LIN {X 0,Y 164.587,Z 329.946,A -85,B 0,C 180,E1 -23658.193,E2 -23658.193} C_VEL
LIN {X 0,Y 167.282,Z 320.465,A -85,B 0,C 180,E1 -23660.938,E2 -23660.938} C_VEL
LIN {X 0,Y 169.157,Z 312.465,A -85,B 0,C 180,E1 -23662.842,E2 -23662.842} C_VEL
LIN {X 0,Y 167.967,Z 302.982,A -85,B 0,C 180,E1 -23665.202,E2 -23665.202} C_VEL
LIN {X 0,Y 166.059,Z 292.21,A -85,B 0,C 180,E1 -23667.577,E2 -23667.577} C_VEL
LIN {X 0,Y 163.931,Z 284.61,A -85,B 0,C 180,E1 -23669.159,E2 -23669.159} C_VEL
LIN {X 0,Y 159.909,Z 273.473,A -85,B 0,C 180,E1 -23671.379,E2 -23671.379} C_VEL
LIN {X 0,Y 158.08,Z 269.283,A -85,B 0,C 180,E1 -23672.192,E2 -23672.192} C_VEL
LIN {X 0,Y 157.989,Z 268.806,A -85,B 0,C 180,E1 -23672.393,E2 -23672.393} C_VEL
LIN {X 0,Y 157.793,Z 268.827,A -85,B 0,C 180,E1 -23677.681,E2 -23677.681} C_VEL
LIN {X 0,Y 157.67,Z 268.846,A -85,B 0,C 180,E1 -23681.32,E2 -23681.32} C_VEL
LIN {X 0,Y 157.48,Z 268.865,A -85,B 0,C 180,E1 -23685.534,E2 -23685.534} C_VEL
LIN {X 0,Y 157.408,Z 268.871,A -85,B 0,C 180,E1 -23690.93,E2 -23690.93} C_VEL
LIN {X 0,Y 157.312,Z 268.897,A -85,B 0,C 180,E1 -23696.692,E2 -23696.692} C_VEL
LIN {X 0,Y 157.277,Z 268.897,A -85,B 0,C 180,E1 -23702.43,E2 -23702.43} C_VEL
LIN {X 0,Y 157.317,Z 268.892,A -85,B 0,C 180,E1 -23706.481,E2 -23706.481} C_VEL
LIN {X 0,Y 157.283,Z 268.893,A -85,B 0,C 180,E1 -23712.09,E2 -23712.09} C_VEL
LIN {X 0,Y 157.299,Z 268.885,A -85,B 0,C 180,E1 -23715.636,E2 -23715.636} C_VEL
LIN {X 0,Y 157.285,Z 268.887,A -85,B 0,C 180,E1 -23721.282,E2 -23721.282} C_VEL
LIN {X 0,Y 157.29,Z 268.867,A -85,B 0,C 180,E1 -23724.494,E2 -23724.494} C_VEL
LIN {X 0,Y 157.294,Z 268.877,A -85,B 0,C 180,E1 -23728.1,E2 -23728.1} C_VEL
LIN {X 0,Y 157.324,Z 268.886,A -85,B 0,C 180,E1 -23733.471,E2 -23733.471} C_VEL
LIN {X 0,Y 157.397,Z 268.851,A -85,B 0,C 180,E1 -23739.673,E2 -23739.673} C_VEL
LIN {X 0,Y 157.478,Z 268.864,A -85,B 0,C 180,E1 -23744.473,E2 -23744.473} C_VEL
LIN {X 0,Y 157.695,Z 268.837,A -85,B 0,C 180,E1 -23749.735,E2 -23749.735} C_VEL
LIN {X 0,Y 157.772,Z 268.814,A -85,B 0,C 180,E1 -23752.324,E2 -23752.324} C_VEL
LIN {X 0,Y 158.263,Z 268.771,A -85,B 0,C 180,E1 -23760.004,E2 -23760.004} C_VEL
LIN {X 0,Y 157.773,Z 268.811,A -85,B 0,C 180,E1 -23767.684,E2 -23767.684} C_VEL
LIN {X 0,Y 157.646,Z 268.843,A -85,B 0,C 180,E1 -23771.24,E2 -23771.24} C_VEL
LIN {X 0,Y 157.463,Z 268.868,A -85,B 0,C 180,E1 -23775.537,E2 -23775.537} C_VEL
LIN {X 0,Y 157.381,Z 268.875,A -85,B 0,C 180,E1 -23780.935,E2 -23780.935} C_VEL
LIN {X 0,Y 157.325,Z 268.88,A -85,B 0,C 180,E1 -23786.686,E2 -23786.686} C_VEL
LIN {X 0,Y 157.3,Z 268.891,A -85,B 0,C 180,E1 -23792.426,E2 -23792.426} C_VEL
LIN {X 0,Y 157.397,Z 268.894,A -85,B 0,C 180,E1 -23794.706,E2 -23794.706} C_VEL
LIN {X 0,Y 158.075,Z 272.801,A -85,B 0,C 180,E1 -23800.899,E2 -23800.899} C_VEL
LIN {X 0,Y 158.59,Z 275.681,A -85,B 0,C 180,E1 -23805.162,E2 -23805.162} C_VEL
LIN {X 0,Y 159.285,Z 279.509,A -85,B 0,C 180,E1 -23810.551,E2 -23810.551} C_VEL
LIN {X 0,Y 161.987,Z 290.335,A -85,B 0,C 180,E1 -23812.106,E2 -23812.106} C_VEL
LIN {X 0,Y 163.705,Z 303.35,A -85,B 0,C 180,E1 -23814.073,E2 -23814.073} C_VEL
LIN {X 0,Y 164.706,Z 315.537,A -85,B 0,C 180,E1 -23816.306,E2 -23816.306} C_VEL
LIN {X 0,Y 165.012,Z 327.489,A -85,B 0,C 180,E1 -23818.905,E2 -23818.905} C_VEL
LIN {X 0,Y 164.792,Z 338.132,A -85,B 0,C 180,E1 -23821.673,E2 -23821.673} C_VEL
LIN {X 0,Y 164.335,Z 342.575,A -85,B 0,C 180,E1 -23822.972,E2 -23822.972} C_VEL
LIN {X 0,Y 161.587,Z 352.064,A -85,B 0,C 180,E1 -23826.068,E2 -23826.068} C_VEL
LIN {X 0,Y 159.321,Z 360.012,A -85,B 0,C 180,E1 -23829.333,E2 -23829.333} C_VEL
LIN {X 0,Y 157.38,Z 367.337,A -85,B 0,C 180,E1 -23833.123,E2 -23833.123} C_VEL
LIN {X 0,Y 155.955,Z 373.175,A -85,B 0,C 180,E1 -23836.976,E2 -23836.976} C_VEL
LIN {X 0,Y 155.267,Z 377.758,A -85,B 0,C 180,E1 -23840.882,E2 -23840.882} C_VEL
LIN {X 0,Y 155.188,Z 381.439,A -85,B 0,C 180,E1 -23845.115,E2 -23845.115} C_VEL
LIN {X 0,Y 155.179,Z 382.901,A -85,B 0,C 180,E1 -23847.402,E2 -23847.402} C_VEL
LIN {X 0,Y 155.293,Z 384.154,A -85,B 0,C 180,E1 -23849.997,E2 -23849.997} C_VEL
LIN {X 0,Y 154.993,Z 385.225,A -85,B 0,C 180,E1 -23853.948,E2 -23853.948} C_VEL
LIN {X 0,Y 155.003,Z 385.398,A -85,B 0,C 180,E1 -23857.815,E2 -23857.815} C_VEL
LIN {X 0,Y 155.909,Z 384.263,A -85,B 0,C 180,E1 -23863.023,E2 -23863.023} C_VEL
LIN {X 0,Y 158.117,Z 381.644,A -85,B 0,C 180,E1 -23868.125,E2 -23868.125} C_VEL
LIN {X 0,Y 161.641,Z 377.372,A -85,B 0,C 180,E1 -23873.033,E2 -23873.033} C_VEL
LIN {X 0,Y 164.907,Z 373.147,A -85,B 0,C 180,E1 -23876.488,E2 -23876.488} C_VEL
LIN {X 0,Y 169.712,Z 366.592,A -85,B 0,C 180,E1 -23880.481,E2 -23880.481} C_VEL
LIN {X 0,Y 174.548,Z 359.672,A -85,B 0,C 180,E1 -23883.614,E2 -23883.614} C_VEL
LIN {X 0,Y 177.754,Z 354.234,A -85,B 0,C 180,E1 -23885.672,E2 -23885.672} C_VEL
LIN {X 0,Y 180.555,Z 346.618,A -85,B 0,C 180,E1 -23888.517,E2 -23888.517} C_VEL
LIN {X 0,Y 182.546,Z 338.652,A -85,B 0,C 180,E1 -23891.297,E2 -23891.297} C_VEL
LIN {X 0,Y 183.154,Z 335.05,A -85,B 0,C 180,E1 -23892.533,E2 -23892.533} C_VEL
LIN {X 0,Y 183.282,Z 332.559,A -85,B 0,C 180,E1 -23893.482,E2 -23893.482} C_VEL
LIN {X 0,Y 182.549,Z 329.462,A -85,B 0,C 180,E1 -23895.048,E2 -23895.048} C_VEL
LIN {X 0,Y 180.077,Z 325.41,A -85,B 0,C 180,E1 -23897.863,E2 -23897.863} C_VEL
LIN {X 0,Y 177.491,Z 320.441,A -85,B 0,C 180,E1 -23901.38,E2 -23901.38} C_VEL
LIN {X 0,Y 176.191,Z 315.483,A -85,B 0,C 180,E1 -23904.536,E2 -23904.536} C_VEL
LIN {X 0,Y 175.099,Z 311.4,A -85,B 0,C 180,E1 -23907.441,E2 -23907.441} C_VEL
LIN {X 0,Y 173.845,Z 307.667,A -85,B 0,C 180,E1 -23910.976,E2 -23910.976} C_VEL
LIN {X 0,Y 173.102,Z 305.534,A -85,B 0,C 180,E1 -23913.47,E2 -23913.47} C_VEL
LIN {X 0,Y 172.072,Z 302.924,A -85,B 0,C 180,E1 -23918.429,E2 -23918.429} C_VEL
LIN {X 0,Y 171.945,Z 302.092,A -85,B 0,C 180,E1 -23920.91,E2 -23920.91} C_VEL
LIN {X 0,Y 171.99,Z 301.706,A -85,B 0,C 180,E1 -23923.375,E2 -23923.375} C_VEL
LIN {X 0,Y 172.781,Z 301.961,A -85,B 0,C 180,E1 -23928.262,E2 -23928.262} C_VEL
LIN {X 0,Y 173.598,Z 302.45,A -85,B 0,C 180,E1 -23930.677,E2 -23930.677} C_VEL
LIN {X 0,Y 174.34,Z 303.735,A -85,B 0,C 180,E1 -23933.05,E2 -23933.05} C_VEL
LIN {X 0,Y 176.32,Z 307.197,A -85,B 0,C 180,E1 -23937.712,E2 -23937.712} C_VEL
LIN {X 0,Y 177.681,Z 311.262,A -85,B 0,C 180,E1 -23941.13,E2 -23941.13} C_VEL
LIN {X 0,Y 179.166,Z 315.803,A -85,B 0,C 180,E1 -23944.496,E2 -23944.496} C_VEL
LIN {X 0,Y 180.317,Z 322.298,A -85,B 0,C 180,E1 -23948.401,E2 -23948.401} C_VEL
LIN {X 0,Y 180.587,Z 327.752,A -85,B 0,C 180,E1 -23951.217,E2 -23951.217} C_VEL
LIN {X 0,Y 179.946,Z 333.811,A -85,B 0,C 180,E1 -23954.125,E2 -23954.125} C_VEL
LIN {X 0,Y 179.697,Z 335.138,A -85,B 0,C 180,E1 -23954.723,E2 -23954.723} C_VEL
LIN {X 0,Y 176.11,Z 341.104,A -85,B 0,C 180,E1 -23956.721,E2 -23956.721} C_VEL
LIN {X 0,Y 171.383,Z 347.887,A -85,B 0,C 180,E1 -23959.416,E2 -23959.416} C_VEL
LIN {X 0,Y 165.978,Z 354.738,A -85,B 0,C 180,E1 -23962.962,E2 -23962.962} C_VEL
LIN {X 0,Y 160.917,Z 360.293,A -85,B 0,C 180,E1 -23966.898,E2 -23966.898} C_VEL
LIN {X 0,Y 156.483,Z 364.662,A -85,B 0,C 180,E1 -23971.429,E2 -23971.429} C_VEL
LIN {X 0,Y 153.937,Z 366.84,A -85,B 0,C 180,E1 -23974.741,E2 -23974.741} C_VEL
LIN {X 0,Y 151.811,Z 368.316,A -85,B 0,C 180,E1 -23978.098,E2 -23978.098} C_VEL
LIN {X 0,Y 150.161,Z 369.099,A -85,B 0,C 180,E1 -23981.513,E2 -23981.513} C_VEL
LIN {X 0,Y 148.898,Z 369.276,A -85,B 0,C 180,E1 -23985.066,E2 -23985.066} C_VEL
LIN {X 0,Y 147.965,Z 368.552,A -85,B 0,C 180,E1 -23989.453,E2 -23989.453} C_VEL
LIN {X 0,Y 147.657,Z 366.732,A -85,B 0,C 180,E1 -23994.004,E2 -23994.004} C_VEL
LIN {X 0,Y 148.074,Z 363.667,A -85,B 0,C 180,E1 -23998.677,E2 -23998.677} C_VEL
LIN {X 0,Y 149.184,Z 359.094,A -85,B 0,C 180,E1 -24003.508,E2 -24003.508} C_VEL
LIN {X 0,Y 150.768,Z 353.195,A -85,B 0,C 180,E1 -24008.107,E2 -24008.107} C_VEL
LIN {X 0,Y 153.045,Z 345.665,A -85,B 0,C 180,E1 -24012.526,E2 -24012.526} C_VEL
LIN {X 0,Y 155.63,Z 337.437,A -85,B 0,C 180,E1 -24016.288,E2 -24016.288} C_VEL
LIN {X 0,Y 158.101,Z 329.265,A -85,B 0,C 180,E1 -24019.267,E2 -24019.267} C_VEL
LIN {X 0,Y 161.001,Z 319.261,A -85,B 0,C 180,E1 -24022.162,E2 -24022.162} C_VEL
LIN {X 0,Y 162.417,Z 313.83,A -85,B 0,C 180,E1 -24023.48,E2 -24023.48} C_VEL
LIN {X 0,Y 161.154,Z 303.303,A -85,B 0,C 180,E1 -24026.252,E2 -24026.252} C_VEL
LIN {X 0,Y 159.17,Z 292.055,A -85,B 0,C 180,E1 -24028.864,E2 -24028.864} C_VEL
LIN {X 0,Y 155.263,Z 279.895,A -85,B 0,C 180,E1 -24031.541,E2 -24031.541} C_VEL
LIN {X 0,Y 152.291,Z 273.166,A -85,B 0,C 180,E1 -24033.025,E2 -24033.025} C_VEL
LIN {X 0,Y 150.941,Z 270.501,A -85,B 0,C 180,E1 -24033.632,E2 -24033.632} C_VEL
LIN {X 0,Y 150.772,Z 269.701,A -85,B 0,C 180,E1 -24033.845,E2 -24033.845} C_VEL
LIN {X 0,Y 150.728,Z 269.706,A -85,B 0,C 180,E1 -24038.044,E2 -24038.044} C_VEL
LIN {X 0,Y 150.601,Z 269.727,A -85,B 0,C 180,E1 -24041.505,E2 -24041.505} C_VEL
LIN {X 0,Y 150.389,Z 269.753,A -85,B 0,C 180,E1 -24046.286,E2 -24046.286} C_VEL
LIN {X 0,Y 150.381,Z 269.747,A -85,B 0,C 180,E1 -24050.836,E2 -24050.836} C_VEL
LIN {X 0,Y 150.241,Z 269.774,A -85,B 0,C 180,E1 -24057.289,E2 -24057.289} C_VEL
LIN {X 0,Y 150.217,Z 269.775,A -85,B 0,C 180,E1 -24062.642,E2 -24062.642} C_VEL
LIN {X 0,Y 150.228,Z 269.773,A -85,B 0,C 180,E1 -24067.461,E2 -24067.461} C_VEL
LIN {X 0,Y 150.224,Z 269.772,A -85,B 0,C 180,E1 -24071.544,E2 -24071.544} C_VEL
LIN {X 0,Y 150.249,Z 269.763,A -85,B 0,C 180,E1 -24075.448,E2 -24075.448} C_VEL
LIN {X 0,Y 150.227,Z 269.771,A -85,B 0,C 180,E1 -24079.09,E2 -24079.09} C_VEL
LIN {X 0,Y 150.234,Z 269.758,A -85,B 0,C 180,E1 -24082.685,E2 -24082.685} C_VEL
LIN {X 0,Y 150.218,Z 269.754,A -85,B 0,C 180,E1 -24087.371,E2 -24087.371} C_VEL
LIN {X 0,Y 150.246,Z 269.769,A -85,B 0,C 180,E1 -24092.723,E2 -24092.723} C_VEL
LIN {X 0,Y 150.354,Z 269.728,A -85,B 0,C 180,E1 -24099.213,E2 -24099.213} C_VEL
LIN {X 0,Y 150.383,Z 269.743,A -85,B 0,C 180,E1 -24103.72,E2 -24103.72} C_VEL
LIN {X 0,Y 150.618,Z 269.72,A -85,B 0,C 180,E1 -24109.247,E2 -24109.247} C_VEL
LIN {X 0,Y 150.709,Z 269.694,A -85,B 0,C 180,E1 -24111.962,E2 -24111.962} C_VEL
LIN {X 0,Y 151.223,Z 269.648,A -85,B 0,C 180,E1 -24120.004,E2 -24120.004} C_VEL
LIN {X 0,Y 150.695,Z 269.692,A -85,B 0,C 180,E1 -24128.047,E2 -24128.047} C_VEL
LIN {X 0,Y 150.587,Z 269.723,A -85,B 0,C 180,E1 -24131.44,E2 -24131.44} C_VEL
LIN {X 0,Y 150.371,Z 269.749,A -85,B 0,C 180,E1 -24136.29,E2 -24136.29} C_VEL
LIN {X 0,Y 150.362,Z 269.749,A -85,B 0,C 180,E1 -24140.795,E2 -24140.795} C_VEL
LIN {X 0,Y 150.255,Z 269.758,A -85,B 0,C 180,E1 -24147.284,E2 -24147.284} C_VEL
LIN {X 0,Y 150.255,Z 269.769,A -85,B 0,C 180,E1 -24152.651,E2 -24152.651} C_VEL
LIN {X 0,Y 150.365,Z 269.919,A -85,B 0,C 180,E1 -24154.526,E2 -24154.526} C_VEL
LIN {X 0,Y 151.01,Z 273.603,A -85,B 0,C 180,E1 -24160.664,E2 -24160.664} C_VEL
LIN {X 0,Y 151.645,Z 277.021,A -85,B 0,C 180,E1 -24165.955,E2 -24165.955} C_VEL
LIN {X 0,Y 152.064,Z 279.225,A -85,B 0,C 180,E1 -24169.04,E2 -24169.04} C_VEL
LIN {X 0,Y 152.993,Z 282.356,A -85,B 0,C 180,E1 -24169.507,E2 -24169.507} C_VEL
LIN {X 0,Y 155.105,Z 289.087,A -85,B 0,C 180,E1 -24170.624,E2 -24170.624} C_VEL
LIN {X 0,Y 156.73,Z 300.075,A -85,B 0,C 180,E1 -24172.371,E2 -24172.371} C_VEL
LIN {X 0,Y 157.918,Z 313.502,A -85,B 0,C 180,E1 -24174.863,E2 -24174.863} C_VEL
LIN {X 0,Y 158.22,Z 324.032,A -85,B 0,C 180,E1 -24177.176,E2 -24177.176} C_VEL
LIN {X 0,Y 158.076,Z 334.837,A -85,B 0,C 180,E1 -24179.986,E2 -24179.986} C_VEL
LIN {X 0,Y 157.685,Z 341.88,A -85,B 0,C 180,E1 -24182.094,E2 -24182.094} C_VEL
LIN {X 0,Y 154.776,Z 351.62,A -85,B 0,C 180,E1 -24185.386,E2 -24185.386} C_VEL
LIN {X 0,Y 152.252,Z 360.086,A -85,B 0,C 180,E1 -24189.036,E2 -24189.036} C_VEL
LIN {X 0,Y 150.256,Z 367.318,A -85,B 0,C 180,E1 -24192.999,E2 -24192.999} C_VEL
LIN {X 0,Y 149.006,Z 372.176,A -85,B 0,C 180,E1 -24196.357,E2 -24196.357} C_VEL
LIN {X 0,Y 148.239,Z 376.889,A -85,B 0,C 180,E1 -24200.446,E2 -24200.446} C_VEL
LIN {X 0,Y 148.124,Z 380.923,A -85,B 0,C 180,E1 -24205.166,E2 -24205.166} C_VEL
LIN {X 0,Y 148.228,Z 383.57,A -85,B 0,C 180,E1 -24209.997,E2 -24209.997} C_VEL
LIN {X 0,Y 147.924,Z 384.692,A -85,B 0,C 180,E1 -24213.809,E2 -24213.809} C_VEL
LIN {X 0,Y 147.953,Z 384.999,A -85,B 0,C 180,E1 -24218.19,E2 -24218.19} C_VEL
LIN {X 0,Y 148.971,Z 383.993,A -85,B 0,C 180,E1 -24223.641,E2 -24223.641} C_VEL
LIN {X 0,Y 151.355,Z 381.5,A -85,B 0,C 180,E1 -24228.965,E2 -24228.965} C_VEL
LIN {X 0,Y 154.044,Z 378.581,A -85,B 0,C 180,E1 -24232.815,E2 -24232.815} C_VEL
LIN {X 0,Y 157.454,Z 374.705,A -85,B 0,C 180,E1 -24236.507,E2 -24236.507} C_VEL
LIN {X 0,Y 161.364,Z 369.808,A -85,B 0,C 180,E1 -24240.054,E2 -24240.054} C_VEL
LIN {X 0,Y 166.955,Z 362.635,A -85,B 0,C 180,E1 -24243.898,E2 -24243.898} C_VEL
LIN {X 0,Y 171.297,Z 356.332,A -85,B 0,C 180,E1 -24246.503,E2 -24246.503} C_VEL
LIN {X 0,Y 174.417,Z 349.2,A -85,B 0,C 180,E1 -24249.351,E2 -24249.351} C_VEL
LIN {X 0,Y 176.905,Z 340.935,A -85,B 0,C 180,E1 -24252.48,E2 -24252.48} C_VEL
LIN {X 0,Y 178.724,Z 331.575,A -85,B 0,C 180,E1 -24255.885,E2 -24255.885} C_VEL
LIN {X 0,Y 178.953,Z 328.046,A -85,B 0,C 180,E1 -24257.271,E2 -24257.271} C_VEL
LIN {X 0,Y 177.746,Z 321.515,A -85,B 0,C 180,E1 -24260.751,E2 -24260.751} C_VEL
LIN {X 0,Y 177.491,Z 320.441,A -85,B 0,C 180,E1 -24261.38,E2 -24261.38} C_VEL
LIN {X 0,Y 176.414,Z 318.23,A -85,B 0,C 180,E1 -24263.116,E2 -24263.116} C_VEL
LIN {X 0,Y 174.799,Z 316.982,A -85,B 0,C 180,E1 -24264.942,E2 -24264.942} C_VEL
LIN {X 0,Y 171.436,Z 315.517,A -85,B 0,C 180,E1 -24268.756,E2 -24268.756} C_VEL
LIN {X 0,Y 170.376,Z 314.318,A -85,B 0,C 180,E1 -24270.707,E2 -24270.707} C_VEL
LIN {X 0,Y 170.201,Z 313.727,A -85,B 0,C 180,E1 -24271.352,E2 -24271.352} C_VEL
LIN {X 0,Y 169.873,Z 312.361,A -85,B 0,C 180,E1 -24272.925,E2 -24272.925} C_VEL
LIN {X 0,Y 169.205,Z 310.428,A -85,B 0,C 180,E1 -24276.027,E2 -24276.027} C_VEL
LIN {X 0,Y 168.8,Z 308.583,A -85,B 0,C 180,E1 -24280.54,E2 -24280.54} C_VEL
LIN {X 0,Y 168.834,Z 308.087,A -85,B 0,C 180,E1 -24283.21,E2 -24283.21} C_VEL
LIN {X 0,Y 169.516,Z 308.242,A -85,B 0,C 180,E1 -24288.032,E2 -24288.032} C_VEL
LIN {X 0,Y 170.259,Z 308.715,A -85,B 0,C 180,E1 -24290.493,E2 -24290.493} C_VEL
LIN {X 0,Y 170.835,Z 309.926,A -85,B 0,C 180,E1 -24292.907,E2 -24292.907} C_VEL
LIN {X 0,Y 172.491,Z 313.333,A -85,B 0,C 180,E1 -24297.661,E2 -24297.661} C_VEL
LIN {X 0,Y 173.9,Z 318.689,A -85,B 0,C 180,E1 -24302.313,E2 -24302.313} C_VEL
LIN {X 0,Y 174.586,Z 321.794,A -85,B 0,C 180,E1 -24304.614,E2 -24304.614} C_VEL
LIN {X 0,Y 175.157,Z 327.207,A -85,B 0,C 180,E1 -24308.069,E2 -24308.069} C_VEL
LIN {X 0,Y 175.059,Z 331.387,A -85,B 0,C 180,E1 -24310.404,E2 -24310.404} C_VEL
LIN {X 0,Y 174.112,Z 337.154,A -85,B 0,C 180,E1 -24313.377,E2 -24313.377} C_VEL
LIN {X 0,Y 171.784,Z 340.942,A -85,B 0,C 180,E1 -24314.726,E2 -24314.726} C_VEL
LIN {X 0,Y 166.076,Z 348.63,A -85,B 0,C 180,E1 -24317.804,E2 -24317.804} C_VEL
LIN {X 0,Y 160.681,Z 355.089,A -85,B 0,C 180,E1 -24321.218,E2 -24321.218} C_VEL
LIN {X 0,Y 155.332,Z 360.626,A -85,B 0,C 180,E1 -24325.196,E2 -24325.196} C_VEL
LIN {X 0,Y 150.443,Z 365.062,A -85,B 0,C 180,E1 -24329.903,E2 -24329.903} C_VEL
LIN {X 0,Y 146.304,Z 368.15,A -85,B 0,C 180,E1 -24335.257,E2 -24335.257} C_VEL
LIN {X 0,Y 143.923,Z 369.385,A -85,B 0,C 180,E1 -24339.4,E2 -24339.4} C_VEL
LIN {X 0,Y 142.14,Z 369.717,A -85,B 0,C 180,E1 -24343.799,E2 -24343.799} C_VEL
LIN {X 0,Y 140.856,Z 368.721,A -85,B 0,C 180,E1 -24349.565,E2 -24349.565} C_VEL
LIN {X 0,Y 140.595,Z 366.413,A -85,B 0,C 180,E1 -24354.914,E2 -24354.914} C_VEL
LIN {X 0,Y 141.224,Z 362.743,A -85,B 0,C 180,E1 -24360.159,E2 -24360.159} C_VEL
LIN {X 0,Y 142.536,Z 357.639,A -85,B 0,C 180,E1 -24365.225,E2 -24365.225} C_VEL
LIN {X 0,Y 144.468,Z 351.073,A -85,B 0,C 180,E1 -24370.094,E2 -24370.094} C_VEL
LIN {X 0,Y 146.814,Z 343.775,A -85,B 0,C 180,E1 -24374.217,E2 -24374.217} C_VEL
LIN {X 0,Y 149.32,Z 335.946,A -85,B 0,C 180,E1 -24377.722,E2 -24377.722} C_VEL
LIN {X 0,Y 152.291,Z 326.599,A -85,B 0,C 180,E1 -24381.042,E2 -24381.042} C_VEL
LIN {X 0,Y 155.444,Z 315.832,A -85,B 0,C 180,E1 -24384.037,E2 -24384.037} C_VEL
LIN {X 0,Y 155.54,Z 312.991,A -85,B 0,C 180,E1 -24384.818,E2 -24384.818} C_VEL
LIN {X 0,Y 154.223,Z 302.636,A -85,B 0,C 180,E1 -24387.657,E2 -24387.657} C_VEL
LIN {X 0,Y 152.425,Z 293.007,A -85,B 0,C 180,E1 -24390.003,E2 -24390.003} C_VEL
LIN {X 0,Y 148.529,Z 280.926,A -85,B 0,C 180,E1 -24392.868,E2 -24392.868} C_VEL
LIN {X 0,Y 144.783,Z 273.65,A -85,B 0,C 180,E1 -24394.745,E2 -24394.745} C_VEL
LIN {X 0,Y 143.71,Z 271.131,A -85,B 0,C 180,E1 -24395.326,E2 -24395.326} C_VEL
LIN {X 0,Y 143.635,Z 270.59,A -85,B 0,C 180,E1 -24395.425,E2 -24395.425} C_VEL
LIN {X 0,Y 143.649,Z 270.586,A -85,B 0,C 180,E1 -24398.443,E2 -24398.443} C_VEL
LIN {X 0,Y 143.538,Z 270.606,A -85,B 0,C 180,E1 -24401.716,E2 -24401.716} C_VEL
LIN {X 0,Y 143.327,Z 270.636,A -85,B 0,C 180,E1 -24407.113,E2 -24407.113} C_VEL
LIN {X 0,Y 143.303,Z 270.626,A -85,B 0,C 180,E1 -24411.294,E2 -24411.294} C_VEL
LIN {X 0,Y 143.187,Z 270.652,A -85,B 0,C 180,E1 -24417.945,E2 -24417.945} C_VEL
LIN {X 0,Y 143.166,Z 270.649,A -85,B 0,C 180,E1 -24423.443,E2 -24423.443} C_VEL
LIN {X 0,Y 143.119,Z 270.653,A -85,B 0,C 180,E1 -24429.674,E2 -24429.674} C_VEL
LIN {X 0,Y 143.158,Z 270.652,A -85,B 0,C 180,E1 -24433.42,E2 -24433.42} C_VEL
LIN {X 0,Y 143.154,Z 270.652,A -85,B 0,C 180,E1 -24437.43,E2 -24437.43} C_VEL
LIN {X 0,Y 143.137,Z 270.647,A -85,B 0,C 180,E1 -24441.78,E2 -24441.78} C_VEL
LIN {X 0,Y 143.185,Z 270.628,A -85,B 0,C 180,E1 -24447.328,E2 -24447.328} C_VEL
LIN {X 0,Y 143.192,Z 270.648,A -85,B 0,C 180,E1 -24452.068,E2 -24452.068} C_VEL
LIN {X 0,Y 143.28,Z 270.61,A -85,B 0,C 180,E1 -24458.751,E2 -24458.751} C_VEL
LIN {X 0,Y 143.318,Z 270.619,A -85,B 0,C 180,E1 -24462.894,E2 -24462.894} C_VEL
LIN {X 0,Y 143.543,Z 270.601,A -85,B 0,C 180,E1 -24468.711,E2 -24468.711} C_VEL
LIN {X 0,Y 143.631,Z 270.578,A -85,B 0,C 180,E1 -24471.563,E2 -24471.563} C_VEL
LIN {X 0,Y 144.182,Z 270.525,A -85,B 0,C 180,E1 -24480.004,E2 -24480.004} C_VEL
LIN {X 0,Y 143.62,Z 270.574,A -85,B 0,C 180,E1 -24488.446,E2 -24488.446} C_VEL
LIN {X 0,Y 143.515,Z 270.605,A -85,B 0,C 180,E1 -24491.633,E2 -24491.633} C_VEL
LIN {X 0,Y 143.311,Z 270.622,A -85,B 0,C 180,E1 -24497.116,E2 -24497.116} C_VEL
LIN {X 0,Y 143.288,Z 270.631,A -85,B 0,C 180,E1 -24501.257,E2 -24501.257} C_VEL
LIN {X 0,Y 143.201,Z 270.636,A -85,B 0,C 180,E1 -24507.939,E2 -24507.939} C_VEL
LIN {X 0,Y 143.292,Z 270.771,A -85,B 0,C 180,E1 -24514.083,E2 -24514.083} C_VEL
LIN {X 0,Y 143.794,Z 273.837,A -85,B 0,C 180,E1 -24519.453,E2 -24519.453} C_VEL
LIN {X 0,Y 144.447,Z 277.118,A -85,B 0,C 180,E1 -24524.873,E2 -24524.873} C_VEL
LIN {X 0,Y 144.754,Z 278.666,A -85,B 0,C 180,E1 -24527.306,E2 -24527.306} C_VEL
LIN {X 0,Y 145.76,Z 281.86,A -85,B 0,C 180,E1 -24527.84,E2 -24527.84} C_VEL
LIN {X 0,Y 148.591,Z 289.961,A -85,B 0,C 180,E1 -24529.373,E2 -24529.373} C_VEL
LIN {X 0,Y 149.988,Z 298.506,A -85,B 0,C 180,E1 -24530.829,E2 -24530.829} C_VEL
LIN {X 0,Y 151.094,Z 311.014,A -85,B 0,C 180,E1 -24533.208,E2 -24533.208} C_VEL
LIN {X 0,Y 151.485,Z 322.367,A -85,B 0,C 180,E1 -24535.766,E2 -24535.766} C_VEL
LIN {X 0,Y 151.385,Z 332.946,A -85,B 0,C 180,E1 -24538.579,E2 -24538.579} C_VEL
LIN {X 0,Y 150.799,Z 342.181,A -85,B 0,C 180,E1 -24541.462,E2 -24541.462} C_VEL
LIN {X 0,Y 147.933,Z 351.262,A -85,B 0,C 180,E1 -24544.683,E2 -24544.683} C_VEL
LIN {X 0,Y 145.204,Z 360.149,A -85,B 0,C 180,E1 -24548.712,E2 -24548.712} C_VEL
LIN {X 0,Y 143.114,Z 367.28,A -85,B 0,C 180,E1 -24552.861,E2 -24552.861} C_VEL
LIN {X 0,Y 141.705,Z 372.94,A -85,B 0,C 180,E1 -24557.101,E2 -24557.101} C_VEL
LIN {X 0,Y 141.064,Z 377.381,A -85,B 0,C 180,E1 -24561.401,E2 -24561.401} C_VEL
LIN {X 0,Y 141.041,Z 380.459,A -85,B 0,C 180,E1 -24565.313,E2 -24565.313} C_VEL
LIN {X 0,Y 141.163,Z 382.984,A -85,B 0,C 180,E1 -24569.997,E2 -24569.997} C_VEL
LIN {X 0,Y 140.854,Z 384.076,A -85,B 0,C 180,E1 -24573.647,E2 -24573.647} C_VEL
LIN {X 0,Y 140.903,Z 384.563,A -85,B 0,C 180,E1 -24578.603,E2 -24578.603} C_VEL
LIN {X 0,Y 142.038,Z 383.729,A -85,B 0,C 180,E1 -24584.321,E2 -24584.321} C_VEL
LIN {X 0,Y 144.632,Z 381.352,A -85,B 0,C 180,E1 -24589.883,E2 -24589.883} C_VEL
LIN {X 0,Y 148.673,Z 377.454,A -85,B 0,C 180,E1 -24595.176,E2 -24595.176} C_VEL
LIN {X 0,Y 152.393,Z 373.399,A -85,B 0,C 180,E1 -24598.958,E2 -24598.958} C_VEL
LIN {X 0,Y 156.85,Z 368.288,A -85,B 0,C 180,E1 -24602.523,E2 -24602.523} C_VEL
LIN {X 0,Y 162.035,Z 361.974,A -85,B 0,C 180,E1 -24605.838,E2 -24605.838} C_VEL
LIN {X 0,Y 165.614,Z 356.974,A -85,B 0,C 180,E1 -24607.972,E2 -24607.972} C_VEL
LIN {X 0,Y 168.671,Z 350.734,A -85,B 0,C 180,E1 -24610.658,E2 -24610.658} C_VEL
LIN {X 0,Y 171.604,Z 342.195,A -85,B 0,C 180,E1 -24614.122,E2 -24614.122} C_VEL
LIN {X 0,Y 173.345,Z 335.147,A -85,B 0,C 180,E1 -24616.865,E2 -24616.865} C_VEL
LIN {X 0,Y 173.759,Z 332.024,A -85,B 0,C 180,E1 -24618.192,E2 -24618.192} C_VEL
LIN {X 0,Y 172.814,Z 325.374,A -85,B 0,C 180,E1 -24622.065,E2 -24622.065} C_VEL
LIN {X 0,Y 171.692,Z 319.866,A -85,B 0,C 180,E1 -24625.876,E2 -24625.876} C_VEL
LIN {X 0,Y 171.255,Z 317.352,A -85,B 0,C 180,E1 -24627.754,E2 -24627.754} C_VEL
LIN {X 0,Y 170.201,Z 313.727,A -85,B 0,C 180,E1 -24631.352,E2 -24631.352} C_VEL
LIN {X 0,Y 169.801,Z 312.828,A -85,B 0,C 180,E1 -24632.629,E2 -24632.629} C_VEL
LIN {X 0,Y 168.744,Z 312.582,A -85,B 0,C 180,E1 -24634.596,E2 -24634.596} C_VEL
LIN {X 0,Y 165.419,Z 314.586,A -85,B 0,C 180,E1 -24640.68,E2 -24640.68} C_VEL
LIN {X 0,Y 165.272,Z 314.522,A -85,B 0,C 180,E1 -24642.08,E2 -24642.08} C_VEL
LIN {X 0,Y 165.918,Z 314.358,A -85,B 0,C 180,E1 -24647.769,E2 -24647.769} C_VEL
LIN {X 0,Y 166.568,Z 314.77,A -85,B 0,C 180,E1 -24650.28,E2 -24650.28} C_VEL
LIN {X 0,Y 167.031,Z 315.932,A -85,B 0,C 180,E1 -24652.745,E2 -24652.745} C_VEL
LIN {X 0,Y 168.351,Z 319.262,A -85,B 0,C 180,E1 -24657.604,E2 -24657.604} C_VEL
LIN {X 0,Y 169.341,Z 324.47,A -85,B 0,C 180,E1 -24662.375,E2 -24662.375} C_VEL
LIN {X 0,Y 169.772,Z 329.295,A -85,B 0,C 180,E1 -24665.938,E2 -24665.938} C_VEL
LIN {X 0,Y 169.642,Z 333.895,A -85,B 0,C 180,E1 -24668.934,E2 -24668.934} C_VEL
LIN {X 0,Y 168.814,Z 338.214,A -85,B 0,C 180,E1 -24671.401,E2 -24671.401} C_VEL
LIN {X 0,Y 168.502,Z 339.377,A -85,B 0,C 180,E1 -24672.033,E2 -24672.033} C_VEL
LIN {X 0,Y 167.589,Z 340.967,A -85,B 0,C 180,E1 -24672.678,E2 -24672.678} C_VEL
LIN {X 0,Y 161.914,Z 348.265,A -85,B 0,C 180,E1 -24675.538,E2 -24675.538} C_VEL
LIN {X 0,Y 156.084,Z 354.892,A -85,B 0,C 180,E1 -24679,E2 -24679} C_VEL
LIN {X 0,Y 151.628,Z 359.331,A -85,B 0,C 180,E1 -24682.035,E2 -24682.035} C_VEL
LIN {X 0,Y 145.739,Z 364.527,A -85,B 0,C 180,E1 -24687.002,E2 -24687.002} C_VEL
LIN {X 0,Y 141.14,Z 367.849,A -85,B 0,C 180,E1 -24692.172,E2 -24692.172} C_VEL
LIN {X 0,Y 137.514,Z 369.746,A -85,B 0,C 180,E1 -24697.821,E2 -24697.821} C_VEL
LIN {X 0,Y 135.178,Z 370.111,A -85,B 0,C 180,E1 -24703.296,E2 -24703.296} C_VEL
LIN {X 0,Y 134.163,Z 369.573,A -85,B 0,C 180,E1 -24707.163,E2 -24707.163} C_VEL
LIN {X 0,Y 133.497,Z 367.956,A -85,B 0,C 180,E1 -24712.147,E2 -24712.147} C_VEL
LIN {X 0,Y 133.685,Z 365.173,A -85,B 0,C 180,E1 -24717.251,E2 -24717.251} C_VEL
LIN {X 0,Y 134.646,Z 360.933,A -85,B 0,C 180,E1 -24722.529,E2 -24722.529} C_VEL
LIN {X 0,Y 135.933,Z 356.247,A -85,B 0,C 180,E1 -24726.89,E2 -24726.89} C_VEL
LIN {X 0,Y 137.908,Z 349.952,A -85,B 0,C 180,E1 -24731.43,E2 -24731.43} C_VEL
LIN {X 0,Y 140.34,Z 342.753,A -85,B 0,C 180,E1 -24735.502,E2 -24735.502} C_VEL
LIN {X 0,Y 143.09,Z 334.555,A -85,B 0,C 180,E1 -24739.183,E2 -24739.183} C_VEL
LIN {X 0,Y 146.108,Z 325.285,A -85,B 0,C 180,E1 -24742.471,E2 -24742.471} C_VEL
LIN {X 0,Y 148.74,Z 316.659,A -85,B 0,C 180,E1 -24744.92,E2 -24744.92} C_VEL
LIN {X 0,Y 148.726,Z 313.206,A -85,B 0,C 180,E1 -24745.938,E2 -24745.938} C_VEL
LIN {X 0,Y 147.516,Z 303.077,A -85,B 0,C 180,E1 -24748.839,E2 -24748.839} C_VEL
LIN {X 0,Y 146.423,Z 296.64,A -85,B 0,C 180,E1 -24750.519,E2 -24750.519} C_VEL
LIN {X 0,Y 142.872,Z 284.784,A -85,B 0,C 180,E1 -24753.599,E2 -24753.599} C_VEL
LIN {X 0,Y 137.946,Z 274.891,A -85,B 0,C 180,E1 -24756.351,E2 -24756.351} C_VEL
LIN {X 0,Y 136.667,Z 272.174,A -85,B 0,C 180,E1 -24757.065,E2 -24757.065} C_VEL
LIN {X 0,Y 136.554,Z 271.475,A -85,B 0,C 180,E1 -24757.21,E2 -24757.21} C_VEL
LIN {X 0,Y 136.481,Z 271.485,A -85,B 0,C 180,E1 -24761.958,E2 -24761.958} C_VEL
LIN {X 0,Y 136.266,Z 271.517,A -85,B 0,C 180,E1 -24768.029,E2 -24768.029} C_VEL
LIN {X 0,Y 136.219,Z 271.507,A -85,B 0,C 180,E1 -24771.785,E2 -24771.785} C_VEL
LIN {X 0,Y 136.113,Z 271.532,A -85,B 0,C 180,E1 -24778.636,E2 -24778.636} C_VEL
LIN {X 0,Y 136.078,Z 271.534,A -85,B 0,C 180,E1 -24784.622,E2 -24784.622} C_VEL
LIN {X 0,Y 136.085,Z 271.529,A -85,B 0,C 180,E1 -24789.234,E2 -24789.234} C_VEL
LIN {X 0,Y 136.094,Z 271.531,A -85,B 0,C 180,E1 -24793.707,E2 -24793.707} C_VEL
LIN {X 0,Y 136.104,Z 271.53,A -85,B 0,C 180,E1 -24797.841,E2 -24797.841} C_VEL
LIN {X 0,Y 136.089,Z 271.525,A -85,B 0,C 180,E1 -24801.711,E2 -24801.711} C_VEL
LIN {X 0,Y 136.091,Z 271.502,A -85,B 0,C 180,E1 -24805.722,E2 -24805.722} C_VEL
LIN {X 0,Y 136.148,Z 271.526,A -85,B 0,C 180,E1 -24812.322,E2 -24812.322} C_VEL
LIN {X 0,Y 136.247,Z 271.484,A -85,B 0,C 180,E1 -24818.839,E2 -24818.839} C_VEL
LIN {X 0,Y 136.283,Z 271.505,A -85,B 0,C 180,E1 -24825.063,E2 -24825.063} C_VEL
LIN {X 0,Y 136.463,Z 271.485,A -85,B 0,C 180,E1 -24828.117,E2 -24828.117} C_VEL
LIN {X 0,Y 136.557,Z 271.462,A -85,B 0,C 180,E1 -24831.123,E2 -24831.123} C_VEL
LIN {X 0,Y 137.139,Z 271.402,A -85,B 0,C 180,E1 -24840.005,E2 -24840.005} C_VEL
LIN {X 0,Y 136.549,Z 271.456,A -85,B 0,C 180,E1 -24848.887,E2 -24848.887} C_VEL
LIN {X 0,Y 136.45,Z 271.486,A -85,B 0,C 180,E1 -24851.894,E2 -24851.894} C_VEL
LIN {X 0,Y 136.252,Z 271.496,A -85,B 0,C 180,E1 -24858.033,E2 -24858.033} C_VEL
LIN {X 0,Y 136.209,Z 271.515,A -85,B 0,C 180,E1 -24861.752,E2 -24861.752} C_VEL
LIN {X 0,Y 136.112,Z 271.521,A -85,B 0,C 180,E1 -24868.618,E2 -24868.618} C_VEL
LIN {X 0,Y 136.222,Z 271.624,A -85,B 0,C 180,E1 -24873.605,E2 -24873.605} C_VEL
LIN {X 0,Y 136.793,Z 274.88,A -85,B 0,C 180,E1 -24879.583,E2 -24879.583} C_VEL
LIN {X 0,Y 137.433,Z 278.178,A -85,B 0,C 180,E1 -24885.269,E2 -24885.269} C_VEL
LIN {X 0,Y 137.638,Z 279.235,A -85,B 0,C 180,E1 -24885.524,E2 -24885.524} C_VEL
LIN {X 0,Y 139.023,Z 282.414,A -85,B 0,C 180,E1 -24886.213,E2 -24886.213} C_VEL
LIN {X 0,Y 142.38,Z 291.903,A -85,B 0,C 180,E1 -24888.21,E2 -24888.21} C_VEL
LIN {X 0,Y 143.617,Z 299.832,A -85,B 0,C 180,E1 -24889.71,E2 -24889.71} C_VEL
LIN {X 0,Y 144.514,Z 311.961,A -85,B 0,C 180,E1 -24892.185,E2 -24892.185} C_VEL
LIN {X 0,Y 144.807,Z 323.611,A -85,B 0,C 180,E1 -24895,E2 -24895} C_VEL
LIN {X 0,Y 144.511,Z 334.334,A -85,B 0,C 180,E1 -24898.067,E2 -24898.067} C_VEL
LIN {X 0,Y 143.921,Z 342.441,A -85,B 0,C 180,E1 -24900.766,E2 -24900.766} C_VEL
LIN {X 0,Y 140.684,Z 352.149,A -85,B 0,C 180,E1 -24904.446,E2 -24904.446} C_VEL
LIN {X 0,Y 138.149,Z 360.19,A -85,B 0,C 180,E1 -24908.354,E2 -24908.354} C_VEL
LIN {X 0,Y 135.989,Z 367.201,A -85,B 0,C 180,E1 -24912.71,E2 -24912.71} C_VEL
LIN {X 0,Y 134.442,Z 373.593,A -85,B 0,C 180,E1 -24917.927,E2 -24917.927} C_VEL
LIN {X 0,Y 133.938,Z 377.777,A -85,B 0,C 180,E1 -24922.459,E2 -24922.459} C_VEL
LIN {X 0,Y 133.963,Z 380.853,A -85,B 0,C 180,E1 -24926.99,E2 -24926.99} C_VEL
LIN {X 0,Y 134.098,Z 382.339,A -85,B 0,C 180,E1 -24929.997,E2 -24929.997} C_VEL
LIN {X 0,Y 133.795,Z 383.461,A -85,B 0,C 180,E1 -24933.533,E2 -24933.533} C_VEL
LIN {X 0,Y 133.856,Z 384.127,A -85,B 0,C 180,E1 -24939.059,E2 -24939.059} C_VEL
LIN {X 0,Y 135.137,Z 383.434,A -85,B 0,C 180,E1 -24945.069,E2 -24945.069} C_VEL
LIN {X 0,Y 136.304,Z 382.527,A -85,B 0,C 180,E1 -24948.018,E2 -24948.018} C_VEL
LIN {X 0,Y 139.901,Z 379.544,A -85,B 0,C 180,E1 -24953.693,E2 -24953.693} C_VEL
LIN {X 0,Y 143.535,Z 376.269,A -85,B 0,C 180,E1 -24957.717,E2 -24957.717} C_VEL
LIN {X 0,Y 147.689,Z 372.018,A -85,B 0,C 180,E1 -24961.561,E2 -24961.561} C_VEL
LIN {X 0,Y 153.538,Z 365.696,A -85,B 0,C 180,E1 -24965.702,E2 -24965.702} C_VEL
LIN {X 0,Y 159.226,Z 358.945,A -85,B 0,C 180,E1 -24968.971,E2 -24968.971} C_VEL
LIN {X 0,Y 162.688,Z 352.868,A -85,B 0,C 180,E1 -24971.749,E2 -24971.749} C_VEL
LIN {X 0,Y 165.89,Z 344.992,A -85,B 0,C 180,E1 -24975.2,E2 -24975.2} C_VEL
LIN {X 0,Y 167.972,Z 338.45,A -85,B 0,C 180,E1 -24977.971,E2 -24977.971} C_VEL
LIN {X 0,Y 168.459,Z 335.773,A -85,B 0,C 180,E1 -24979.198,E2 -24979.198} C_VEL
LIN {X 0,Y 168.019,Z 330.33,A -85,B 0,C 180,E1 -24982.627,E2 -24982.627} C_VEL
LIN {X 0,Y 167.196,Z 324.614,A -85,B 0,C 180,E1 -24986.872,E2 -24986.872} C_VEL
LIN {X 0,Y 167.051,Z 322.891,A -85,B 0,C 180,E1 -24988.267,E2 -24988.267} C_VEL
LIN {X 0,Y 166.16,Z 318.764,A -85,B 0,C 180,E1 -24992.646,E2 -24992.646} C_VEL
LIN {X 0,Y 165.428,Z 315.919,A -85,B 0,C 180,E1 -24997.517,E2 -24997.517} C_VEL
LIN {X 0,Y 165.272,Z 314.522,A -85,B 0,C 180,E1 -25002.08,E2 -25002.08} C_VEL
LIN {X 0,Y 165.144,Z 314.725,A -85,B 0,C 180,E1 -25004.124,E2 -25004.124} C_VEL
LIN {X 0,Y 164.596,Z 315.933,A -85,B 0,C 180,E1 -25006.136,E2 -25006.136} C_VEL
LIN {X 0,Y 162.99,Z 320.905,A -85,B 0,C 180,E1 -25011.478,E2 -25011.478} C_VEL
LIN {X 0,Y 162.982,Z 321.895,A -85,B 0,C 180,E1 -25012.856,E2 -25012.856} C_VEL
LIN {X 0,Y 163.92,Z 324.961,A -85,B 0,C 180,E1 -25017.539,E2 -25017.539} C_VEL
LIN {X 0,Y 164.456,Z 330.035,A -85,B 0,C 180,E1 -25022.445,E2 -25022.445} C_VEL
LIN {X 0,Y 164.432,Z 334.686,A -85,B 0,C 180,E1 -25026.13,E2 -25026.13} C_VEL
LIN {X 0,Y 163.907,Z 338.368,A -85,B 0,C 180,E1 -25028.628,E2 -25028.628} C_VEL
LIN {X 0,Y 163.02,Z 341.491,A -85,B 0,C 180,E1 -25030.554,E2 -25030.554} C_VEL
LIN {X 0,Y 161.394,Z 343.885,A -85,B 0,C 180,E1 -25031.562,E2 -25031.562} C_VEL
LIN {X 0,Y 154.616,Z 351.749,A -85,B 0,C 180,E1 -25035.014,E2 -25035.014} C_VEL
LIN {X 0,Y 148.417,Z 357.951,A -85,B 0,C 180,E1 -25038.736,E2 -25038.736} C_VEL
LIN {X 0,Y 142.214,Z 363.304,A -85,B 0,C 180,E1 -25043.283,E2 -25043.283} C_VEL
LIN {X 0,Y 137.873,Z 366.505,A -85,B 0,C 180,E1 -25047.302,E2 -25047.302} C_VEL
LIN {X 0,Y 133.463,Z 369.135,A -85,B 0,C 180,E1 -25052.596,E2 -25052.596} C_VEL
LIN {X 0,Y 131.019,Z 370.18,A -85,B 0,C 180,E1 -25056.432,E2 -25056.432} C_VEL
LIN {X 0,Y 128.875,Z 370.56,A -85,B 0,C 180,E1 -25060.867,E2 -25060.867} C_VEL
LIN {X 0,Y 127.311,Z 370.064,A -85,B 0,C 180,E1 -25065.853,E2 -25065.853} C_VEL
LIN {X 0,Y 126.42,Z 368.037,A -85,B 0,C 180,E1 -25072.305,E2 -25072.305} C_VEL
LIN {X 0,Y 126.711,Z 364.647,A -85,B 0,C 180,E1 -25078.292,E2 -25078.292} C_VEL
LIN {X 0,Y 127.869,Z 360.014,A -85,B 0,C 180,E1 -25083.919,E2 -25083.919} C_VEL
LIN {X 0,Y 129.404,Z 354.845,A -85,B 0,C 180,E1 -25088.605,E2 -25088.605} C_VEL
LIN {X 0,Y 131.831,Z 347.598,A -85,B 0,C 180,E1 -25093.638,E2 -25093.638} C_VEL
LIN {X 0,Y 134.704,Z 339.532,A -85,B 0,C 180,E1 -25097.957,E2 -25097.957} C_VEL
LIN {X 0,Y 138.024,Z 329.949,A -85,B 0,C 180,E1 -25101.954,E2 -25101.954} C_VEL
LIN {X 0,Y 141.081,Z 320.511,A -85,B 0,C 180,E1 -25105.015,E2 -25105.015} C_VEL
LIN {X 0,Y 142.218,Z 316.595,A -85,B 0,C 180,E1 -25106.112,E2 -25106.112} C_VEL
LIN {X 0,Y 141.19,Z 306.069,A -85,B 0,C 180,E1 -25109.389,E2 -25109.389} C_VEL
LIN {X 0,Y 139.896,Z 298.32,A -85,B 0,C 180,E1 -25111.625,E2 -25111.625} C_VEL
LIN {X 0,Y 136.968,Z 288.086,A -85,B 0,C 180,E1 -25114.49,E2 -25114.49} C_VEL
LIN {X 0,Y 130.927,Z 275.787,A -85,B 0,C 180,E1 -25118.242,E2 -25118.242} C_VEL
LIN {X 0,Y 129.62,Z 272.89,A -85,B 0,C 180,E1 -25119.069,E2 -25119.069} C_VEL
LIN {X 0,Y 129.505,Z 272.346,A -85,B 0,C 180,E1 -25119.274,E2 -25119.274} C_VEL
LIN {X 0,Y 129.385,Z 272.368,A -85,B 0,C 180,E1 -25122.552,E2 -25122.552} C_VEL
LIN {X 0,Y 129.178,Z 272.398,A -85,B 0,C 180,E1 -25129.056,E2 -25129.056} C_VEL
LIN {X 0,Y 129.128,Z 272.391,A -85,B 0,C 180,E1 -25132.398,E2 -25132.398} C_VEL
LIN {X 0,Y 129.029,Z 272.416,A -85,B 0,C 180,E1 -25139.379,E2 -25139.379} C_VEL
LIN {X 0,Y 129.02,Z 272.416,A -85,B 0,C 180,E1 -25145.215,E2 -25145.215} C_VEL
LIN {X 0,Y 129.01,Z 272.414,A -85,B 0,C 180,E1 -25150.826,E2 -25150.826} C_VEL
LIN {X 0,Y 129.022,Z 272.407,A -85,B 0,C 180,E1 -25155.087,E2 -25155.087} C_VEL
LIN {X 0,Y 129.012,Z 272.414,A -85,B 0,C 180,E1 -25159.704,E2 -25159.704} C_VEL
LIN {X 0,Y 129.023,Z 272.382,A -85,B 0,C 180,E1 -25164.797,E2 -25164.797} C_VEL
LIN {X 0,Y 129.034,Z 272.409,A -85,B 0,C 180,E1 -25170.653,E2 -25170.653} C_VEL
LIN {X 0,Y 129.111,Z 272.38,A -85,B 0,C 180,E1 -25177.608,E2 -25177.608} C_VEL
LIN {X 0,Y 129.162,Z 272.366,A -85,B 0,C 180,E1 -25180.95,E2 -25180.95} C_VEL
LIN {X 0,Y 129.404,Z 272.365,A -85,B 0,C 180,E1 -25187.861,E2 -25187.861} C_VEL
LIN {X 0,Y 129.485,Z 272.346,A -85,B 0,C 180,E1 -25190.634,E2 -25190.634} C_VEL
LIN {X 0,Y 130.094,Z 272.279,A -85,B 0,C 180,E1 -25200.005,E2 -25200.005} C_VEL
LIN {X 0,Y 129.475,Z 272.339,A -85,B 0,C 180,E1 -25209.377,E2 -25209.377} C_VEL
LIN {X 0,Y 129.354,Z 272.372,A -85,B 0,C 180,E1 -25212.557,E2 -25212.557} C_VEL
LIN {X 0,Y 129.163,Z 272.378,A -85,B 0,C 180,E1 -25219.06,E2 -25219.06} C_VEL
LIN {X 0,Y 129.119,Z 272.401,A -85,B 0,C 180,E1 -25222.401,E2 -25222.401} C_VEL
LIN {X 0,Y 129.047,Z 272.404,A -85,B 0,C 180,E1 -25229.376,E2 -25229.376} C_VEL
LIN {X 0,Y 129.171,Z 272.396,A -85,B 0,C 180,E1 -25232.968,E2 -25232.968} C_VEL
LIN {X 0,Y 129.639,Z 275.238,A -85,B 0,C 180,E1 -25238.573,E2 -25238.573} C_VEL
LIN {X 0,Y 130.143,Z 277.802,A -85,B 0,C 180,E1 -25243.252,E2 -25243.252} C_VEL
LIN {X 0,Y 131.156,Z 280.969,A -85,B 0,C 180,E1 -25243.894,E2 -25243.894} C_VEL
LIN {X 0,Y 132.328,Z 283.66,A -85,B 0,C 180,E1 -25244.549,E2 -25244.549} C_VEL
LIN {X 0,Y 135.542,Z 292.079,A -85,B 0,C 180,E1 -25246.551,E2 -25246.551} C_VEL
LIN {X 0,Y 136.911,Z 297.477,A -85,B 0,C 180,E1 -25247.745,E2 -25247.745} C_VEL
LIN {X 0,Y 137.896,Z 310.177,A -85,B 0,C 180,E1 -25250.451,E2 -25250.451} C_VEL
LIN {X 0,Y 138.164,Z 322.003,A -85,B 0,C 180,E1 -25253.402,E2 -25253.402} C_VEL
LIN {X 0,Y 137.783,Z 333.292,A -85,B 0,C 180,E1 -25256.744,E2 -25256.744} C_VEL
LIN {X 0,Y 137.042,Z 342.564,A -85,B 0,C 180,E1 -25259.996,E2 -25259.996} C_VEL
LIN {X 0,Y 133.764,Z 352.066,A -85,B 0,C 180,E1 -25263.797,E2 -25263.797} C_VEL
LIN {X 0,Y 131.1,Z 360.151,A -85,B 0,C 180,E1 -25267.957,E2 -25267.957} C_VEL
LIN {X 0,Y 128.884,Z 367.073,A -85,B 0,C 180,E1 -25272.544,E2 -25272.544} C_VEL
LIN {X 0,Y 127.483,Z 372.605,A -85,B 0,C 180,E1 -25277.257,E2 -25277.257} C_VEL
LIN {X 0,Y 126.888,Z 376.924,A -85,B 0,C 180,E1 -25282.038,E2 -25282.038} C_VEL
LIN {X 0,Y 126.886,Z 380.129,A -85,B 0,C 180,E1 -25286.822,E2 -25286.822} C_VEL
LIN {X 0,Y 127.033,Z 381.677,A -85,B 0,C 180,E1 -25289.997,E2 -25289.997} C_VEL
LIN {X 0,Y 126.749,Z 382.854,A -85,B 0,C 180,E1 -25293.497,E2 -25293.497} C_VEL
LIN {X 0,Y 126.834,Z 383.691,A -85,B 0,C 180,E1 -25299.566,E2 -25299.566} C_VEL
LIN {X 0,Y 128.246,Z 383.121,A -85,B 0,C 180,E1 -25305.899,E2 -25305.899} C_VEL
LIN {X 0,Y 131.325,Z 381.1,A -85,B 0,C 180,E1 -25311.997,E2 -25311.997} C_VEL
LIN {X 0,Y 135.927,Z 377.483,A -85,B 0,C 180,E1 -25317.729,E2 -25317.729} C_VEL
LIN {X 0,Y 140.112,Z 373.726,A -85,B 0,C 180,E1 -25321.778,E2 -25321.778} C_VEL
LIN {X 0,Y 145.085,Z 368.953,A -85,B 0,C 180,E1 -25325.538,E2 -25325.538} C_VEL
LIN {X 0,Y 151.826,Z 361.915,A -85,B 0,C 180,E1 -25329.527,E2 -25329.527} C_VEL
LIN {X 0,Y 154.615,Z 358.39,A -85,B 0,C 180,E1 -25331.227,E2 -25331.227} C_VEL
LIN {X 0,Y 158.129,Z 352.17,A -85,B 0,C 180,E1 -25334.267,E2 -25334.267} C_VEL
LIN {X 0,Y 161.441,Z 344.682,A -85,B 0,C 180,E1 -25337.733,E2 -25337.733} C_VEL
LIN {X 0,Y 162.93,Z 340.404,A -85,B 0,C 180,E1 -25339.678,E2 -25339.678} C_VEL
LIN {X 0,Y 163.09,Z 336.971,A -85,B 0,C 180,E1 -25341.881,E2 -25341.881} C_VEL
LIN {X 0,Y 162.775,Z 331.652,A -85,B 0,C 180,E1 -25345.851,E2 -25345.851} C_VEL
LIN {X 0,Y 162.564,Z 328.261,A -85,B 0,C 180,E1 -25348.745,E2 -25348.745} C_VEL
LIN {X 0,Y 162.056,Z 324.618,A -85,B 0,C 180,E1 -25352.794,E2 -25352.794} C_VEL
LIN {X 0,Y 161.548,Z 322.198,A -85,B 0,C 180,E1 -25356.946,E2 -25356.946} C_VEL
LIN {X 0,Y 161.475,Z 321.124,A -85,B 0,C 180,E1 -25359.62,E2 -25359.62} C_VEL
LIN {X 0,Y 161.523,Z 320.337,A -85,B 0,C 180,E1 -25363.174,E2 -25363.174} C_VEL
LIN {X 0,Y 161.987,Z 320.287,A -85,B 0,C 180,E1 -25367.467,E2 -25367.467} C_VEL
LIN {X 0,Y 162.567,Z 320.624,A -85,B 0,C 180,E1 -25370.038,E2 -25370.038} C_VEL
LIN {X 0,Y 162.982,Z 321.895,A -85,B 0,C 180,E1 -25372.856,E2 -25372.856} C_VEL
LIN {X 0,Y 162.886,Z 323.668,A -85,B 0,C 180,E1 -25374.839,E2 -25374.839} C_VEL
LIN {X 0,Y 162.243,Z 326.222,A -85,B 0,C 180,E1 -25376.716,E2 -25376.716} C_VEL
LIN {X 0,Y 159.511,Z 334.155,A -85,B 0,C 180,E1 -25381.642,E2 -25381.642} C_VEL
LIN {X 0,Y 159.184,Z 335.822,A -85,B 0,C 180,E1 -25382.958,E2 -25382.958} C_VEL
LIN {X 0,Y 158.699,Z 339.892,A -85,B 0,C 180,E1 -25386.352,E2 -25386.352} C_VEL
LIN {X 0,Y 157.744,Z 343.179,A -85,B 0,C 180,E1 -25388.658,E2 -25388.658} C_VEL
LIN {X 0,Y 156.821,Z 344.922,A -85,B 0,C 180,E1 -25389.636,E2 -25389.636} C_VEL
LIN {X 0,Y 149.62,Z 352.693,A -85,B 0,C 180,E1 -25393.131,E2 -25393.131} C_VEL
LIN {X 0,Y 142.631,Z 359.17,A -85,B 0,C 180,E1 -25397.191,E2 -25397.191} C_VEL
LIN {X 0,Y 136.207,Z 364.199,A -85,B 0,C 180,E1 -25401.766,E2 -25401.766} C_VEL
LIN {X 0,Y 132.201,Z 366.934,A -85,B 0,C 180,E1 -25405.352,E2 -25405.352} C_VEL
LIN {X 0,Y 128.381,Z 369.074,A -85,B 0,C 180,E1 -25409.511,E2 -25409.511} C_VEL
LIN {X 0,Y 125.007,Z 370.478,A -85,B 0,C 180,E1 -25414.202,E2 -25414.202} C_VEL
LIN {X 0,Y 122.373,Z 370.984,A -85,B 0,C 180,E1 -25419.171,E2 -25419.171} C_VEL
LIN {X 0,Y 120.264,Z 370.363,A -85,B 0,C 180,E1 -25425.477,E2 -25425.477} C_VEL
LIN {X 0,Y 119.513,Z 369.111,A -85,B 0,C 180,E1 -25429.851,E2 -25429.851} C_VEL
LIN {X 0,Y 119.338,Z 366.522,A -85,B 0,C 180,E1 -25435.525,E2 -25435.525} C_VEL
LIN {X 0,Y 120.282,Z 361.98,A -85,B 0,C 180,E1 -25442.136,E2 -25442.136} C_VEL
LIN {X 0,Y 121.784,Z 356.919,A -85,B 0,C 180,E1 -25447.404,E2 -25447.404} C_VEL
LIN {X 0,Y 124.033,Z 350.254,A -85,B 0,C 180,E1 -25452.697,E2 -25452.697} C_VEL
LIN {X 0,Y 126.71,Z 342.966,A -85,B 0,C 180,E1 -25457.185,E2 -25457.185} C_VEL
LIN {X 0,Y 129.986,Z 334.059,A -85,B 0,C 180,E1 -25461.452,E2 -25461.452} C_VEL
LIN {X 0,Y 133.675,Z 323.527,A -85,B 0,C 180,E1 -25465.318,E2 -25465.318} C_VEL
LIN {X 0,Y 135.479,Z 317.865,A -85,B 0,C 180,E1 -25467.029,E2 -25467.029} C_VEL
LIN {X 0,Y 134.685,Z 307.752,A -85,B 0,C 180,E1 -25470.377,E2 -25470.377} C_VEL
LIN {X 0,Y 133.64,Z 301.056,A -85,B 0,C 180,E1 -25472.433,E2 -25472.433} C_VEL
LIN {X 0,Y 130.832,Z 290.941,A -85,B 0,C 180,E1 -25475.547,E2 -25475.547} C_VEL
LIN {X 0,Y 125.621,Z 279.963,A -85,B 0,C 180,E1 -25479.259,E2 -25479.259} C_VEL
LIN {X 0,Y 123.779,Z 276.623,A -85,B 0,C 180,E1 -25480.415,E2 -25480.415} C_VEL
LIN {X 0,Y 122.498,Z 273.991,A -85,B 0,C 180,E1 -25481.266,E2 -25481.266} C_VEL
LIN {X 0,Y 122.357,Z 273.245,A -85,B 0,C 180,E1 -25481.523,E2 -25481.523} C_VEL
LIN {X 0,Y 122.123,Z 273.275,A -85,B 0,C 180,E1 -25486.726,E2 -25486.726} C_VEL
LIN {X 0,Y 122.06,Z 273.272,A -85,B 0,C 180,E1 -25492.906,E2 -25492.906} C_VEL
LIN {X 0,Y 121.955,Z 273.298,A -85,B 0,C 180,E1 -25497.457,E2 -25497.457} C_VEL
LIN {X 0,Y 121.907,Z 273.305,A -85,B 0,C 180,E1 -25501.259,E2 -25501.259} C_VEL
LIN {X 0,Y 121.933,Z 273.299,A -85,B 0,C 180,E1 -25506.213,E2 -25506.213} C_VEL
LIN {X 0,Y 121.939,Z 273.296,A -85,B 0,C 180,E1 -25511.482,E2 -25511.482} C_VEL
LIN {X 0,Y 121.94,Z 273.297,A -85,B 0,C 180,E1 -25518.531,E2 -25518.531} C_VEL
LIN {X 0,Y 121.975,Z 273.259,A -85,B 0,C 180,E1 -25524.824,E2 -25524.824} C_VEL
LIN {X 0,Y 121.943,Z 273.288,A -85,B 0,C 180,E1 -25529.833,E2 -25529.833} C_VEL
LIN {X 0,Y 121.986,Z 273.277,A -85,B 0,C 180,E1 -25536.222,E2 -25536.222} C_VEL
LIN {X 0,Y 122.051,Z 273.247,A -85,B 0,C 180,E1 -25539.794,E2 -25539.794} C_VEL
LIN {X 0,Y 122.249,Z 273.256,A -85,B 0,C 180,E1 -25546.711,E2 -25546.711} C_VEL
LIN {X 0,Y 122.421,Z 273.227,A -85,B 0,C 180,E1 -25550.088,E2 -25550.088} C_VEL
LIN {X 0,Y 122.602,Z 273.193,A -85,B 0,C 180,E1 -25556.719,E2 -25556.719} C_VEL
LIN {X 0,Y 123.047,Z 273.157,A -85,B 0,C 180,E1 -25560.005,E2 -25560.005} C_VEL
LIN {X 0,Y 122.425,Z 273.211,A -85,B 0,C 180,E1 -25566.598,E2 -25566.598} C_VEL
LIN {X 0,Y 122.321,Z 273.248,A -85,B 0,C 180,E1 -25572.368,E2 -25572.368} C_VEL
LIN {X 0,Y 122.118,Z 273.263,A -85,B 0,C 180,E1 -25576.729,E2 -25576.729} C_VEL
LIN {X 0,Y 122.035,Z 273.284,A -85,B 0,C 180,E1 -25582.854,E2 -25582.854} C_VEL
LIN {X 0,Y 122.015,Z 273.285,A -85,B 0,C 180,E1 -25590.226,E2 -25590.226} C_VEL
LIN {X 0,Y 122.127,Z 273.334,A -85,B 0,C 180,E1 -25592.655,E2 -25592.655} C_VEL
LIN {X 0,Y 122.664,Z 276.438,A -85,B 0,C 180,E1 -25599.074,E2 -25599.074} C_VEL
LIN {X 0,Y 122.858,Z 277.302,A -85,B 0,C 180,E1 -25600.806,E2 -25600.806} C_VEL
LIN {X 0,Y 123.892,Z 280.53,A -85,B 0,C 180,E1 -25601.539,E2 -25601.539} C_VEL
LIN {X 0,Y 125.133,Z 283.12,A -85,B 0,C 180,E1 -25602.283,E2 -25602.283} C_VEL
LIN {X 0,Y 129.121,Z 293.431,A -85,B 0,C 180,E1 -25605.045,E2 -25605.045} C_VEL
LIN {X 0,Y 130.697,Z 299.486,A -85,B 0,C 180,E1 -25606.553,E2 -25606.553} C_VEL
LIN {X 0,Y 131.473,Z 311.864,A -85,B 0,C 180,E1 -25609.395,E2 -25609.395} C_VEL
LIN {X 0,Y 131.549,Z 323.416,A -85,B 0,C 180,E1 -25612.52,E2 -25612.52} C_VEL
LIN {X 0,Y 130.974,Z 334.78,A -85,B 0,C 180,E1 -25616.167,E2 -25616.167} C_VEL
LIN {X 0,Y 130.193,Z 342.687,A -85,B 0,C 180,E1 -25619.144,E2 -25619.144} C_VEL
LIN {X 0,Y 126.872,Z 351.965,A -85,B 0,C 180,E1 -25623.068,E2 -25623.068} C_VEL
LIN {X 0,Y 124.046,Z 360.093,A -85,B 0,C 180,E1 -25627.512,E2 -25627.512} C_VEL
LIN {X 0,Y 121.778,Z 366.945,A -85,B 0,C 180,E1 -25632.36,E2 -25632.36} C_VEL
LIN {X 0,Y 120.214,Z 373.223,A -85,B 0,C 180,E1 -25638.189,E2 -25638.189} C_VEL
LIN {X 0,Y 119.78,Z 377.295,A -85,B 0,C 180,E1 -25643.258,E2 -25643.258} C_VEL
LIN {X 0,Y 119.821,Z 379.399,A -85,B 0,C 180,E1 -25646.634,E2 -25646.634} C_VEL
LIN {X 0,Y 119.968,Z 381.004,A -85,B 0,C 180,E1 -25649.997,E2 -25649.997} C_VEL
LIN {X 0,Y 119.691,Z 382.139,A -85,B 0,C 180,E1 -25653.363,E2 -25653.363} C_VEL
LIN {X 0,Y 119.806,Z 383.245,A -85,B 0,C 180,E1 -25660.132,E2 -25660.132} C_VEL
LIN {X 0,Y 121.388,Z 382.808,A -85,B 0,C 180,E1 -25666.824,E2 -25666.824} C_VEL
LIN {X 0,Y 124.755,Z 380.932,A -85,B 0,C 180,E1 -25673.221,E2 -25673.221} C_VEL
LIN {X 0,Y 126.986,Z 379.444,A -85,B 0,C 180,E1 -25676.276,E2 -25676.276} C_VEL
LIN {X 0,Y 132.189,Z 375.504,A -85,B 0,C 180,E1 -25681.709,E2 -25681.709} C_VEL
LIN {X 0,Y 137.539,Z 370.945,A -85,B 0,C 180,E1 -25685.985,E2 -25685.985} C_VEL
LIN {X 0,Y 144.35,Z 364.593,A -85,B 0,C 180,E1 -25690.17,E2 -25690.17} C_VEL
LIN {X 0,Y 148.447,Z 360.265,A -85,B 0,C 180,E1 -25692.423,E2 -25692.423} C_VEL
LIN {X 0,Y 151.877,Z 355.122,A -85,B 0,C 180,E1 -25695.137,E2 -25695.137} C_VEL
LIN {X 0,Y 155.239,Z 348.809,A -85,B 0,C 180,E1 -25698.326,E2 -25698.326} C_VEL
LIN {X 0,Y 157.034,Z 344.88,A -85,B 0,C 180,E1 -25700.246,E2 -25700.246} C_VEL
LIN {X 0,Y 157.615,Z 342.906,A -85,B 0,C 180,E1 -25701.368,E2 -25701.368} C_VEL
LIN {X 0,Y 157.8,Z 338.614,A -85,B 0,C 180,E1 -25704.617,E2 -25704.617} C_VEL
LIN {X 0,Y 157.833,Z 333.619,A -85,B 0,C 180,E1 -25709.026,E2 -25709.026} C_VEL
LIN {X 0,Y 157.614,Z 329.85,A -85,B 0,C 180,E1 -25713.515,E2 -25713.515} C_VEL
LIN {X 0,Y 157.373,Z 328.258,A -85,B 0,C 180,E1 -25716.298,E2 -25716.298} C_VEL
LIN {X 0,Y 157.292,Z 326.867,A -85,B 0,C 180,E1 -25719.761,E2 -25719.761} C_VEL
LIN {X 0,Y 157.449,Z 326.035,A -85,B 0,C 180,E1 -25724.462,E2 -25724.462} C_VEL
LIN {X 0,Y 158.259,Z 326.29,A -85,B 0,C 180,E1 -25729.764,E2 -25729.764} C_VEL
LIN {X 0,Y 158.582,Z 327.372,A -85,B 0,C 180,E1 -25732.5,E2 -25732.5} C_VEL
LIN {X 0,Y 159.199,Z 330.429,A -85,B 0,C 180,E1 -25737.466,E2 -25737.466} C_VEL
LIN {X 0,Y 159.256,Z 334.002,A -85,B 0,C 180,E1 -25741.26,E2 -25741.26} C_VEL
LIN {X 0,Y 159.184,Z 335.822,A -85,B 0,C 180,E1 -25742.958,E2 -25742.958} C_VEL
LIN {X 0,Y 158.651,Z 337.651,A -85,B 0,C 180,E1 -25744.206,E2 -25744.206} C_VEL
LIN {X 0,Y 156.738,Z 340.969,A -85,B 0,C 180,E1 -25745.853,E2 -25745.853} C_VEL
LIN {X 0,Y 153.935,Z 344.57,A -85,B 0,C 180,E1 -25747.297,E2 -25747.297} C_VEL
LIN {X 0,Y 149.322,Z 349.412,A -85,B 0,C 180,E1 -25749.159,E2 -25749.159} C_VEL
LIN {X 0,Y 144.655,Z 353.82,A -85,B 0,C 180,E1 -25751.211,E2 -25751.211} C_VEL
LIN {X 0,Y 138.117,Z 359.484,A -85,B 0,C 180,E1 -25754.816,E2 -25754.816} C_VEL
LIN {X 0,Y 132.387,Z 363.74,A -85,B 0,C 180,E1 -25758.568,E2 -25758.568} C_VEL
LIN {X 0,Y 127.214,Z 367.044,A -85,B 0,C 180,E1 -25762.745,E2 -25762.745} C_VEL
LIN {X 0,Y 122.722,Z 369.404,A -85,B 0,C 180,E1 -25767.261,E2 -25767.261} C_VEL
LIN {X 0,Y 118.046,Z 371.129,A -85,B 0,C 180,E1 -25773.546,E2 -25773.546} C_VEL
LIN {X 0,Y 115.729,Z 371.418,A -85,B 0,C 180,E1 -25777.87,E2 -25777.87} C_VEL
LIN {X 0,Y 113.866,Z 371.041,A -85,B 0,C 180,E1 -25782.752,E2 -25782.752} C_VEL
LIN {X 0,Y 112.558,Z 369.669,A -85,B 0,C 180,E1 -25788.518,E2 -25788.518} C_VEL
LIN {X 0,Y 112.26,Z 366.554,A -85,B 0,C 180,E1 -25795.71,E2 -25795.71} C_VEL
LIN {X 0,Y 113.237,Z 361.96,A -85,B 0,C 180,E1 -25802.531,E2 -25802.531} C_VEL
LIN {X 0,Y 114.979,Z 356.384,A -85,B 0,C 180,E1 -25808.489,E2 -25808.489} C_VEL
LIN {X 0,Y 117.208,Z 350.14,A -85,B 0,C 180,E1 -25813.593,E2 -25813.593} C_VEL
LIN {X 0,Y 119.963,Z 342.983,A -85,B 0,C 180,E1 -25818.171,E2 -25818.171} C_VEL
LIN {X 0,Y 123.399,Z 333.968,A -85,B 0,C 180,E1 -25822.641,E2 -25822.641} C_VEL
LIN {X 0,Y 126.773,Z 324.792,A -85,B 0,C 180,E1 -25826.178,E2 -25826.178} C_VEL
LIN {X 0,Y 128.831,Z 318.065,A -85,B 0,C 180,E1 -25828.36,E2 -25828.36} C_VEL
LIN {X 0,Y 128.026,Z 307.769,A -85,B 0,C 180,E1 -25831.968,E2 -25831.968} C_VEL
LIN {X 0,Y 126.817,Z 301.456,A -85,B 0,C 180,E1 -25834.109,E2 -25834.109} C_VEL
LIN {X 0,Y 125.013,Z 294.462,A -85,B 0,C 180,E1 -25836.459,E2 -25836.459} C_VEL
LIN {X 0,Y 119.801,Z 283.169,A -85,B 0,C 180,E1 -25840.63,E2 -25840.63} C_VEL
LIN {X 0,Y 116.779,Z 277.677,A -85,B 0,C 180,E1 -25842.779,E2 -25842.779} C_VEL
LIN {X 0,Y 115.364,Z 275.144,A -85,B 0,C 180,E1 -25843.777,E2 -25843.777} C_VEL
LIN {X 0,Y 115.143,Z 274.134,A -85,B 0,C 180,E1 -25844.135,E2 -25844.135} C_VEL
LIN {X 0,Y 115.005,Z 274.149,A -85,B 0,C 180,E1 -25851.514,E2 -25851.514} C_VEL
LIN {X 0,Y 114.874,Z 274.183,A -85,B 0,C 180,E1 -25855.361,E2 -25855.361} C_VEL
LIN {X 0,Y 114.864,Z 274.183,A -85,B 0,C 180,E1 -25861.075,E2 -25861.075} C_VEL
LIN {X 0,Y 114.844,Z 274.181,A -85,B 0,C 180,E1 -25867.736,E2 -25867.736} C_VEL
LIN {X 0,Y 114.862,Z 274.178,A -85,B 0,C 180,E1 -25872.766,E2 -25872.766} C_VEL
LIN {X 0,Y 114.867,Z 274.176,A -85,B 0,C 180,E1 -25877.708,E2 -25877.708} C_VEL
LIN {X 0,Y 114.854,Z 274.16,A -85,B 0,C 180,E1 -25882.706,E2 -25882.706} C_VEL
LIN {X 0,Y 114.869,Z 274.163,A -85,B 0,C 180,E1 -25888.939,E2 -25888.939} C_VEL
LIN {X 0,Y 114.949,Z 274.151,A -85,B 0,C 180,E1 -25896.514,E2 -25896.514} C_VEL
LIN {X 0,Y 115.02,Z 274.134,A -85,B 0,C 180,E1 -25902.217,E2 -25902.217} C_VEL
LIN {X 0,Y 115.258,Z 274.127,A -85,B 0,C 180,E1 -25907.337,E2 -25907.337} C_VEL
LIN {X 0,Y 115.371,Z 274.083,A -85,B 0,C 180,E1 -25913.008,E2 -25913.008} C_VEL
LIN {X 0,Y 115.999,Z 274.034,A -85,B 0,C 180,E1 -25920.005,E2 -25920.005} C_VEL
LIN {X 0,Y 115.367,Z 274.088,A -85,B 0,C 180,E1 -25927.004,E2 -25927.004} C_VEL
LIN {X 0,Y 115.258,Z 274.128,A -85,B 0,C 180,E1 -25932.662,E2 -25932.662} C_VEL
LIN {X 0,Y 115.021,Z 274.14,A -85,B 0,C 180,E1 -25937.794,E2 -25937.794} C_VEL
LIN {X 0,Y 114.958,Z 274.168,A -85,B 0,C 180,E1 -25943.496,E2 -25943.496} C_VEL
LIN {X 0,Y 115.045,Z 274.155,A -85,B 0,C 180,E1 -25952.078,E2 -25952.078} C_VEL
LIN {X 0,Y 115.532,Z 277.078,A -85,B 0,C 180,E1 -25958.093,E2 -25958.093} C_VEL
LIN {X 0,Y 116.808,Z 280.499,A -85,B 0,C 180,E1 -25959.031,E2 -25959.031} C_VEL
LIN {X 0,Y 117.883,Z 282.601,A -85,B 0,C 180,E1 -25959.725,E2 -25959.725} C_VEL
LIN {X 0,Y 120.916,Z 289.724,A -85,B 0,C 180,E1 -25961.875,E2 -25961.875} C_VEL
LIN {X 0,Y 123.77,Z 298.295,A -85,B 0,C 180,E1 -25964.376,E2 -25964.376} C_VEL
LIN {X 0,Y 124.706,Z 303.372,A -85,B 0,C 180,E1 -25965.722,E2 -25965.722} C_VEL
LIN {X 0,Y 125.055,Z 314.904,A -85,B 0,C 180,E1 -25968.67,E2 -25968.67} C_VEL
LIN {X 0,Y 124.863,Z 326.092,A -85,B 0,C 180,E1 -25972.006,E2 -25972.006} C_VEL
LIN {X 0,Y 124.009,Z 337.282,A -85,B 0,C 180,E1 -25975.965,E2 -25975.965} C_VEL
LIN {X 0,Y 123.404,Z 342.763,A -85,B 0,C 180,E1 -25978.207,E2 -25978.207} C_VEL
LIN {X 0,Y 120.128,Z 351.467,A -85,B 0,C 180,E1 -25982.09,E2 -25982.09} C_VEL
LIN {X 0,Y 117.032,Z 359.978,A -85,B 0,C 180,E1 -25987.021,E2 -25987.021} C_VEL
LIN {X 0,Y 114.685,Z 366.765,A -85,B 0,C 180,E1 -25992.154,E2 -25992.154} C_VEL
LIN {X 0,Y 113.255,Z 372.184,A -85,B 0,C 180,E1 -25997.452,E2 -25997.452} C_VEL
LIN {X 0,Y 112.728,Z 376.4,A -85,B 0,C 180,E1 -26002.834,E2 -26002.834} C_VEL
LIN {X 0,Y 112.766,Z 378.604,A -85,B 0,C 180,E1 -26006.423,E2 -26006.423} C_VEL
LIN {X 0,Y 112.905,Z 380.317,A -85,B 0,C 180,E1 -26009.996,E2 -26009.996} C_VEL
LIN {X 0,Y 112.611,Z 381.513,A -85,B 0,C 180,E1 -26013.575,E2 -26013.575} C_VEL
LIN {X 0,Y 112.807,Z 382.749,A -85,B 0,C 180,E1 -26020.768,E2 -26020.768} C_VEL
LIN {X 0,Y 114.568,Z 382.501,A -85,B 0,C 180,E1 -26027.858,E2 -26027.858} C_VEL
LIN {X 0,Y 118.235,Z 380.767,A -85,B 0,C 180,E1 -26034.584,E2 -26034.584} C_VEL
LIN {X 0,Y 123.483,Z 377.564,A -85,B 0,C 180,E1 -26040.809,E2 -26040.809} C_VEL
LIN {X 0,Y 130.011,Z 372.708,A -85,B 0,C 180,E1 -26046.482,E2 -26046.482} C_VEL
LIN {X 0,Y 135.815,Z 367.929,A -85,B 0,C 180,E1 -26050.3,E2 -26050.3} C_VEL
LIN {X 0,Y 142.271,Z 362.007,A -85,B 0,C 180,E1 -26053.751,E2 -26053.751} C_VEL
LIN {X 0,Y 145.811,Z 357.508,A -85,B 0,C 180,E1 -26056.298,E2 -26056.298} C_VEL
LIN {X 0,Y 149.7,Z 351.268,A -85,B 0,C 180,E1 -26059.716,E2 -26059.716} C_VEL
LIN {X 0,Y 151.801,Z 347.226,A -85,B 0,C 180,E1 -26061.907,E2 -26061.907} C_VEL
LIN {X 0,Y 152.35,Z 344.507,A -85,B 0,C 180,E1 -26063.969,E2 -26063.969} C_VEL
LIN {X 0,Y 152.707,Z 340.337,A -85,B 0,C 180,E1 -26067.752,E2 -26067.752} C_VEL
LIN {X 0,Y 152.866,Z 338.427,A -85,B 0,C 180,E1 -26069.616,E2 -26069.616} C_VEL
LIN {X 0,Y 152.885,Z 336.005,A -85,B 0,C 180,E1 -26072.629,E2 -26072.629} C_VEL
LIN {X 0,Y 152.796,Z 333.496,A -85,B 0,C 180,E1 -26076.908,E2 -26076.908} C_VEL
LIN {X 0,Y 152.828,Z 332.049,A -85,B 0,C 180,E1 -26081.218,E2 -26081.218} C_VEL
LIN {X 0,Y 153.228,Z 331.539,A -85,B 0,C 180,E1 -26086.738,E2 -26086.738} C_VEL
LIN {X 0,Y 153.674,Z 331.73,A -85,B 0,C 180,E1 -26089.455,E2 -26089.455} C_VEL
LIN {X 0,Y 153.917,Z 332.599,A -85,B 0,C 180,E1 -26092.123,E2 -26092.123} C_VEL
LIN {X 0,Y 154.017,Z 333.94,A -85,B 0,C 180,E1 -26094.76,E2 -26094.76} C_VEL
LIN {X 0,Y 154.2,Z 335.624,A -85,B 0,C 180,E1 -26097.384,E2 -26097.384} C_VEL
LIN {X 0,Y 153.909,Z 339.056,A -85,B 0,C 180,E1 -26101.304,E2 -26101.304} C_VEL
LIN {X 0,Y 153.124,Z 343.253,A -85,B 0,C 180,E1 -26105.263,E2 -26105.263} C_VEL
LIN {X 0,Y 152.209,Z 345.801,A -85,B 0,C 180,E1 -26107.291,E2 -26107.291} C_VEL
LIN {X 0,Y 151.51,Z 346.924,A -85,B 0,C 180,E1 -26107.995,E2 -26107.995} C_VEL
LIN {X 0,Y 144.655,Z 353.82,A -85,B 0,C 180,E1 -26111.211,E2 -26111.211} C_VEL
LIN {X 0,Y 141.053,Z 356.753,A -85,B 0,C 180,E1 -26112.688,E2 -26112.688} C_VEL
LIN {X 0,Y 133.84,Z 361.229,A -85,B 0,C 180,E1 -26114.841,E2 -26114.841} C_VEL
LIN {X 0,Y 126.662,Z 365.01,A -85,B 0,C 180,E1 -26117.338,E2 -26117.338} C_VEL
LIN {X 0,Y 123.22,Z 366.767,A -85,B 0,C 180,E1 -26119.359,E2 -26119.359} C_VEL
LIN {X 0,Y 117.293,Z 369.75,A -85,B 0,C 180,E1 -26124.792,E2 -26124.792} C_VEL
LIN {X 0,Y 113.109,Z 371.239,A -85,B 0,C 180,E1 -26129.8,E2 -26129.8} C_VEL
LIN {X 0,Y 109.748,Z 371.84,A -85,B 0,C 180,E1 -26135.186,E2 -26135.186} C_VEL
LIN {X 0,Y 107.285,Z 371.525,A -85,B 0,C 180,E1 -26140.917,E2 -26140.917} C_VEL
LIN {X 0,Y 105.488,Z 369.825,A -85,B 0,C 180,E1 -26148.228,E2 -26148.228} C_VEL
LIN {X 0,Y 105.172,Z 366.732,A -85,B 0,C 180,E1 -26155.558,E2 -26155.558} C_VEL
LIN {X 0,Y 106.046,Z 362.392,A -85,B 0,C 180,E1 -26162.365,E2 -26162.365} C_VEL
LIN {X 0,Y 107.948,Z 356.535,A -85,B 0,C 180,E1 -26169.022,E2 -26169.022} C_VEL
LIN {X 0,Y 110.317,Z 350.212,A -85,B 0,C 180,E1 -26174.457,E2 -26174.457} C_VEL
LIN {X 0,Y 113.226,Z 343,A -85,B 0,C 180,E1 -26179.272,E2 -26179.272} C_VEL
LIN {X 0,Y 116.866,Z 333.879,A -85,B 0,C 180,E1 -26183.962,E2 -26183.962} C_VEL
LIN {X 0,Y 120.784,Z 323.65,A -85,B 0,C 180,E1 -26187.989,E2 -26187.989} C_VEL
LIN {X 0,Y 122.063,Z 320.008,A -85,B 0,C 180,E1 -26189.179,E2 -26189.179} C_VEL
LIN {X 0,Y 121.905,Z 313.601,A -85,B 0,C 180,E1 -26191.646,E2 -26191.646} C_VEL
LIN {X 0,Y 121.364,Z 307.646,A -85,B 0,C 180,E1 -26193.809,E2 -26193.809} C_VEL
LIN {X 0,Y 119.272,Z 298.413,A -85,B 0,C 180,E1 -26197.196,E2 -26197.196} C_VEL
LIN {X 0,Y 114.73,Z 287.849,A -85,B 0,C 180,E1 -26201.477,E2 -26201.477} C_VEL
LIN {X 0,Y 110.786,Z 280.534,A -85,B 0,C 180,E1 -26204.703,E2 -26204.703} C_VEL
LIN {X 0,Y 108.298,Z 276.379,A -85,B 0,C 180,E1 -26206.614,E2 -26206.614} C_VEL
LIN {X 0,Y 107.981,Z 275.038,A -85,B 0,C 180,E1 -26207.033,E2 -26207.033} C_VEL
LIN {X 0,Y 107.866,Z 275.049,A -85,B 0,C 180,E1 -26214.209,E2 -26214.209} C_VEL
LIN {X 0,Y 107.794,Z 275.062,A -85,B 0,C 180,E1 -26222.063,E2 -26222.063} C_VEL
LIN {X 0,Y 107.751,Z 275.06,A -85,B 0,C 180,E1 -26228.502,E2 -26228.502} C_VEL
LIN {X 0,Y 107.766,Z 275.054,A -85,B 0,C 180,E1 -26235.843,E2 -26235.843} C_VEL
LIN {X 0,Y 107.754,Z 275.053,A -85,B 0,C 180,E1 -26241.512,E2 -26241.512} C_VEL
LIN {X 0,Y 107.811,Z 275.039,A -85,B 0,C 180,E1 -26248.574,E2 -26248.574} C_VEL
LIN {X 0,Y 107.913,Z 275.021,A -85,B 0,C 180,E1 -26257.005,E2 -26257.005} C_VEL
LIN {X 0,Y 108.038,Z 275.022,A -85,B 0,C 180,E1 -26264.924,E2 -26264.924} C_VEL
LIN {X 0,Y 108.263,Z 274.996,A -85,B 0,C 180,E1 -26268.776,E2 -26268.776} C_VEL
LIN {X 0,Y 108.45,Z 274.949,A -85,B 0,C 180,E1 -26276.29,E2 -26276.29} C_VEL
LIN {X 0,Y 108.948,Z 274.912,A -85,B 0,C 180,E1 -26280.006,E2 -26280.006} C_VEL
LIN {X 0,Y 108.307,Z 274.965,A -85,B 0,C 180,E1 -26287.463,E2 -26287.463} C_VEL
LIN {X 0,Y 108.179,Z 275.01,A -85,B 0,C 180,E1 -26292.953,E2 -26292.953} C_VEL
LIN {X 0,Y 107.914,Z 275.023,A -85,B 0,C 180,E1 -26299.01,E2 -26299.01} C_VEL
LIN {X 0,Y 107.869,Z 275.049,A -85,B 0,C 180,E1 -26304.188,E2 -26304.188} C_VEL
LIN {X 0,Y 108.003,Z 275.123,A -85,B 0,C 180,E1 -26311.87,E2 -26311.87} C_VEL
LIN {X 0,Y 108.176,Z 276.34,A -85,B 0,C 180,E1 -26314.777,E2 -26314.777} C_VEL
LIN {X 0,Y 109.186,Z 279.473,A -85,B 0,C 180,E1 -26315.698,E2 -26315.698} C_VEL
LIN {X 0,Y 110.773,Z 282.269,A -85,B 0,C 180,E1 -26316.836,E2 -26316.836} C_VEL
LIN {X 0,Y 114.255,Z 290.44,A -85,B 0,C 180,E1 -26319.663,E2 -26319.663} C_VEL
LIN {X 0,Y 117.69,Z 300.609,A -85,B 0,C 180,E1 -26322.968,E2 -26322.968} C_VEL
LIN {X 0,Y 118.538,Z 305.036,A -85,B 0,C 180,E1 -26324.285,E2 -26324.285} C_VEL
LIN {X 0,Y 118.656,Z 316.204,A -85,B 0,C 180,E1 -26327.375,E2 -26327.375} C_VEL
LIN {X 0,Y 118.299,Z 326.151,A -85,B 0,C 180,E1 -26330.57,E2 -26330.57} C_VEL
LIN {X 0,Y 117.296,Z 337.293,A -85,B 0,C 180,E1 -26334.777,E2 -26334.777} C_VEL
LIN {X 0,Y 116.624,Z 342.747,A -85,B 0,C 180,E1 -26337.152,E2 -26337.152} C_VEL
LIN {X 0,Y 113.226,Z 351.392,A -85,B 0,C 180,E1 -26341.242,E2 -26341.242} C_VEL
LIN {X 0,Y 110.01,Z 359.825,A -85,B 0,C 180,E1 -26346.463,E2 -26346.463} C_VEL
LIN {X 0,Y 107.583,Z 366.564,A -85,B 0,C 180,E1 -26351.919,E2 -26351.919} C_VEL
LIN {X 0,Y 105.983,Z 372.739,A -85,B 0,C 180,E1 -26358.521,E2 -26358.521} C_VEL
LIN {X 0,Y 105.658,Z 376.726,A -85,B 0,C 180,E1 -26364.272,E2 -26364.272} C_VEL
LIN {X 0,Y 105.843,Z 379.593,A -85,B 0,C 180,E1 -26369.996,E2 -26369.996} C_VEL
LIN {X 0,Y 105.534,Z 380.884,A -85,B 0,C 180,E1 -26373.815,E2 -26373.815} C_VEL
LIN {X 0,Y 105.808,Z 382.24,A -85,B 0,C 180,E1 -26381.49,E2 -26381.49} C_VEL
LIN {X 0,Y 107.796,Z 382.155,A -85,B 0,C 180,E1 -26389.021,E2 -26389.021} C_VEL
LIN {X 0,Y 111.78,Z 380.602,A -85,B 0,C 180,E1 -26396.107,E2 -26396.107} C_VEL
LIN {X 0,Y 117.406,Z 377.562,A -85,B 0,C 180,E1 -26402.594,E2 -26402.594} C_VEL
LIN {X 0,Y 122.489,Z 374.255,A -85,B 0,C 180,E1 -26407.042,E2 -26407.042} C_VEL
LIN {X 0,Y 128.38,Z 369.987,A -85,B 0,C 180,E1 -26411.061,E2 -26411.061} C_VEL
LIN {X 0,Y 136.149,Z 363.642,A -85,B 0,C 180,E1 -26415.212,E2 -26415.212} C_VEL
LIN {X 0,Y 139.135,Z 360.516,A -85,B 0,C 180,E1 -26417.086,E2 -26417.086} C_VEL
LIN {X 0,Y 143.28,Z 355.037,A -85,B 0,C 180,E1 -26420.378,E2 -26420.378} C_VEL
LIN {X 0,Y 145.851,Z 351.069,A -85,B 0,C 180,E1 -26422.657,E2 -26422.657} C_VEL
LIN {X 0,Y 146.726,Z 348.66,A -85,B 0,C 180,E1 -26424.511,E2 -26424.511} C_VEL
LIN {X 0,Y 147.483,Z 344.119,A -85,B 0,C 180,E1 -26429.06,E2 -26429.06} C_VEL
LIN {X 0,Y 147.735,Z 341.973,A -85,B 0,C 180,E1 -26431.59,E2 -26431.59} C_VEL
LIN {X 0,Y 147.868,Z 339.975,A -85,B 0,C 180,E1 -26434.67,E2 -26434.67} C_VEL
LIN {X 0,Y 147.973,Z 338.492,A -85,B 0,C 180,E1 -26437.664,E2 -26437.664} C_VEL
LIN {X 0,Y 148.096,Z 337.276,A -85,B 0,C 180,E1 -26441.634,E2 -26441.634} C_VEL
LIN {X 0,Y 148.425,Z 336.835,A -85,B 0,C 180,E1 -26446.301,E2 -26446.301} C_VEL
LIN {X 0,Y 148.815,Z 336.919,A -85,B 0,C 180,E1 -26449.107,E2 -26449.107} C_VEL
LIN {X 0,Y 148.971,Z 337.8,A -85,B 0,C 180,E1 -26452.166,E2 -26452.166} C_VEL
LIN {X 0,Y 148.952,Z 338.932,A -85,B 0,C 180,E1 -26454.581,E2 -26454.581} C_VEL
LIN {X 0,Y 148.918,Z 340.545,A -85,B 0,C 180,E1 -26457.291,E2 -26457.291} C_VEL
LIN {X 0,Y 148.257,Z 343.839,A -85,B 0,C 180,E1 -26461.354,E2 -26461.354} C_VEL
LIN {X 0,Y 147.506,Z 346.508,A -85,B 0,C 180,E1 -26464.093,E2 -26464.093} C_VEL
LIN {X 0,Y 146.523,Z 348.751,A -85,B 0,C 180,E1 -26466.097,E2 -26466.097} C_VEL
LIN {X 0,Y 138.522,Z 356.083,A -85,B 0,C 180,E1 -26469.823,E2 -26469.823} C_VEL
LIN {X 0,Y 130.513,Z 362.225,A -85,B 0,C 180,E1 -26474.251,E2 -26474.251} C_VEL
LIN {X 0,Y 123.22,Z 366.767,A -85,B 0,C 180,E1 -26479.359,E2 -26479.359} C_VEL
LIN {X 0,Y 119.894,Z 368.374,A -85,B 0,C 180,E1 -26481.541,E2 -26481.541} C_VEL
LIN {X 0,Y 113.216,Z 370.512,A -85,B 0,C 180,E1 -26484.996,E2 -26484.996} C_VEL
LIN {X 0,Y 108.031,Z 371.646,A -85,B 0,C 180,E1 -26488.06,E2 -26488.06} C_VEL
LIN {X 0,Y 105.002,Z 372.132,A -85,B 0,C 180,E1 -26490.781,E2 -26490.781} C_VEL
LIN {X 0,Y 104.279,Z 372.196,A -85,B 0,C 180,E1 -26491.784,E2 -26491.784} C_VEL
LIN {X 0,Y 100.79,Z 372.002,A -85,B 0,C 180,E1 -26498.862,E2 -26498.862} C_VEL
LIN {X 0,Y 98.878,Z 370.759,A -85,B 0,C 180,E1 -26505.288,E2 -26505.288} C_VEL
LIN {X 0,Y 98.029,Z 368.426,A -85,B 0,C 180,E1 -26512.046,E2 -26512.046} C_VEL
LIN {X 0,Y 98.352,Z 364.846,A -85,B 0,C 180,E1 -26519.022,E2 -26519.022} C_VEL
LIN {X 0,Y 99.856,Z 359.718,A -85,B 0,C 180,E1 -26526.183,E2 -26526.183} C_VEL
LIN {X 0,Y 102.211,Z 353.305,A -85,B 0,C 180,E1 -26532.826,E2 -26532.826} C_VEL
LIN {X 0,Y 105.599,Z 345.094,A -85,B 0,C 180,E1 -26539.115,E2 -26539.115} C_VEL
LIN {X 0,Y 108.776,Z 337.626,A -85,B 0,C 180,E1 -26543.512,E2 -26543.512} C_VEL
LIN {X 0,Y 112.792,Z 327.906,A -85,B 0,C 180,E1 -26547.959,E2 -26547.959} C_VEL
LIN {X 0,Y 115.434,Z 321.033,A -85,B 0,C 180,E1 -26550.434,E2 -26550.434} C_VEL
LIN {X 0,Y 115.389,Z 314.666,A -85,B 0,C 180,E1 -26553.041,E2 -26553.041} C_VEL
LIN {X 0,Y 114.656,Z 307.973,A -85,B 0,C 180,E1 -26555.691,E2 -26555.691} C_VEL
LIN {X 0,Y 112.947,Z 300.62,A -85,B 0,C 180,E1 -26558.681,E2 -26558.681} C_VEL
LIN {X 0,Y 109.126,Z 291.451,A -85,B 0,C 180,E1 -26562.819,E2 -26562.819} C_VEL
LIN {X 0,Y 105.405,Z 284.444,A -85,B 0,C 180,E1 -26566.252,E2 -26566.252} C_VEL
LIN {X 0,Y 103.456,Z 280.961,A -85,B 0,C 180,E1 -26568.024,E2 -26568.024} C_VEL
LIN {X 0,Y 101.218,Z 277.488,A -85,B 0,C 180,E1 -26569.984,E2 -26569.984} C_VEL
LIN {X 0,Y 100.814,Z 275.919,A -85,B 0,C 180,E1 -26570.67,E2 -26570.67} C_VEL
LIN {X 0,Y 100.767,Z 275.938,A -85,B 0,C 180,E1 -26574.965,E2 -26574.965} C_VEL
LIN {X 0,Y 100.702,Z 275.94,A -85,B 0,C 180,E1 -26583.138,E2 -26583.138} C_VEL
LIN {X 0,Y 100.698,Z 275.937,A -85,B 0,C 180,E1 -26589.861,E2 -26589.861} C_VEL
LIN {X 0,Y 100.732,Z 275.93,A -85,B 0,C 180,E1 -26595.768,E2 -26595.768} C_VEL
LIN {X 0,Y 100.694,Z 275.934,A -85,B 0,C 180,E1 -26601.094,E2 -26601.094} C_VEL
LIN {X 0,Y 100.707,Z 275.908,A -85,B 0,C 180,E1 -26606.877,E2 -26606.877} C_VEL
LIN {X 0,Y 100.788,Z 275.921,A -85,B 0,C 180,E1 -26615.275,E2 -26615.275} C_VEL
LIN {X 0,Y 100.82,Z 275.888,A -85,B 0,C 180,E1 -26619.609,E2 -26619.609} C_VEL
LIN {X 0,Y 101.108,Z 275.89,A -85,B 0,C 180,E1 -26626.706,E2 -26626.706} C_VEL
LIN {X 0,Y 101.25,Z 275.846,A -85,B 0,C 180,E1 -26632.026,E2 -26632.026} C_VEL
LIN {X 0,Y 101.872,Z 275.794,A -85,B 0,C 180,E1 -26640.006,E2 -26640.006} C_VEL
LIN {X 0,Y 101.246,Z 275.844,A -85,B 0,C 180,E1 -26647.986,E2 -26647.986} C_VEL
LIN {X 0,Y 101.109,Z 275.891,A -85,B 0,C 180,E1 -26653.296,E2 -26653.296} C_VEL
LIN {X 0,Y 100.826,Z 275.91,A -85,B 0,C 180,E1 -26660.403,E2 -26660.403} C_VEL
LIN {X 0,Y 100.786,Z 275.928,A -85,B 0,C 180,E1 -26664.962,E2 -26664.962} C_VEL
LIN {X 0,Y 100.904,Z 276.097,A -85,B 0,C 180,E1 -26671.061,E2 -26671.061} C_VEL
LIN {X 0,Y 102.16,Z 279.283,A -85,B 0,C 180,E1 -26672.263,E2 -26672.263} C_VEL
LIN {X 0,Y 103.509,Z 281.678,A -85,B 0,C 180,E1 -26673.374,E2 -26673.374} C_VEL
LIN {X 0,Y 105.473,Z 285.798,A -85,B 0,C 180,E1 -26675.086,E2 -26675.086} C_VEL
LIN {X 0,Y 108.93,Z 294.479,A -85,B 0,C 180,E1 -26678.395,E2 -26678.395} C_VEL
LIN {X 0,Y 111.777,Z 303.653,A -85,B 0,C 180,E1 -26681.742,E2 -26681.742} C_VEL
LIN {X 0,Y 112.371,Z 308.031,A -85,B 0,C 180,E1 -26683.138,E2 -26683.138} C_VEL
LIN {X 0,Y 112.148,Z 320.086,A -85,B 0,C 180,E1 -26686.853,E2 -26686.853} C_VEL
LIN {X 0,Y 111.464,Z 329.638,A -85,B 0,C 180,E1 -26690.276,E2 -26690.276} C_VEL
LIN {X 0,Y 110.345,Z 339.591,A -85,B 0,C 180,E1 -26694.462,E2 -26694.462} C_VEL
LIN {X 0,Y 109.887,Z 342.612,A -85,B 0,C 180,E1 -26695.906,E2 -26695.906} C_VEL
LIN {X 0,Y 106.345,Z 351.314,A -85,B 0,C 180,E1 -26700.283,E2 -26700.283} C_VEL
LIN {X 0,Y 102.995,Z 359.665,A -85,B 0,C 180,E1 -26705.827,E2 -26705.827} C_VEL
LIN {X 0,Y 100.494,Z 366.349,A -85,B 0,C 180,E1 -26711.653,E2 -26711.653} C_VEL
LIN {X 0,Y 99.014,Z 371.673,A -85,B 0,C 180,E1 -26717.701,E2 -26717.701} C_VEL
LIN {X 0,Y 98.606,Z 375.808,A -85,B 0,C 180,E1 -26723.859,E2 -26723.859} C_VEL
LIN {X 0,Y 98.781,Z 378.814,A -85,B 0,C 180,E1 -26729.996,E2 -26729.996} C_VEL
LIN {X 0,Y 98.475,Z 380.19,A -85,B 0,C 180,E1 -26734.088,E2 -26734.088} C_VEL
LIN {X 0,Y 98.428,Z 381.162,A -85,B 0,C 180,E1 -26738.206,E2 -26738.206} C_VEL
LIN {X 0,Y 99.707,Z 381.934,A -85,B 0,C 180,E1 -26746.372,E2 -26746.372} C_VEL
LIN {X 0,Y 103.03,Z 381.287,A -85,B 0,C 180,E1 -26754.155,E2 -26754.155} C_VEL
LIN {X 0,Y 108.259,Z 379.199,A -85,B 0,C 180,E1 -26761.284,E2 -26761.284} C_VEL
LIN {X 0,Y 115.005,Z 375.567,A -85,B 0,C 180,E1 -26767.665,E2 -26767.665} C_VEL
LIN {X 0,Y 120.95,Z 371.794,A -85,B 0,C 180,E1 -26771.926,E2 -26771.926} C_VEL
LIN {X 0,Y 127.666,Z 367.035,A -85,B 0,C 180,E1 -26775.691,E2 -26775.691} C_VEL
LIN {X 0,Y 132.349,Z 363.262,A -85,B 0,C 180,E1 -26778.019,E2 -26778.019} C_VEL
LIN {X 0,Y 136.157,Z 359.153,A -85,B 0,C 180,E1 -26780.733,E2 -26780.733} C_VEL
LIN {X 0,Y 139.735,Z 354.59,A -85,B 0,C 180,E1 -26783.579,E2 -26783.579} C_VEL
LIN {X 0,Y 140.846,Z 352.778,A -85,B 0,C 180,E1 -26784.898,E2 -26784.898} C_VEL
LIN {X 0,Y 141.869,Z 348.949,A -85,B 0,C 180,E1 -26788.968,E2 -26788.968} C_VEL
LIN {X 0,Y 142.45,Z 346.173,A -85,B 0,C 180,E1 -26792.624,E2 -26792.624} C_VEL
LIN {X 0,Y 142.741,Z 343.89,A -85,B 0,C 180,E1 -26796.799,E2 -26796.799} C_VEL
LIN {X 0,Y 142.926,Z 342.807,A -85,B 0,C 180,E1 -26799.862,E2 -26799.862} C_VEL
LIN {X 0,Y 143.102,Z 342.112,A -85,B 0,C 180,E1 -26802.858,E2 -26802.858} C_VEL
LIN {X 0,Y 143.661,Z 341.863,A -85,B 0,C 180,E1 -26808.711,E2 -26808.711} C_VEL
LIN {X 0,Y 143.81,Z 342.474,A -85,B 0,C 180,E1 -26811.565,E2 -26811.565} C_VEL
LIN {X 0,Y 143.662,Z 343.67,A -85,B 0,C 180,E1 -26814.381,E2 -26814.381} C_VEL
LIN {X 0,Y 143.39,Z 345.201,A -85,B 0,C 180,E1 -26817.186,E2 -26817.186} C_VEL
LIN {X 0,Y 142.346,Z 348.378,A -85,B 0,C 180,E1 -26821.41,E2 -26821.41} C_VEL
LIN {X 0,Y 141.881,Z 349.613,A -85,B 0,C 180,E1 -26822.835,E2 -26822.835} C_VEL
LIN {X 0,Y 140.98,Z 351.226,A -85,B 0,C 180,E1 -26824.463,E2 -26824.463} C_VEL
LIN {X 0,Y 134.603,Z 356.63,A -85,B 0,C 180,E1 -26827.259,E2 -26827.259} C_VEL
LIN {X 0,Y 125.864,Z 362.897,A -85,B 0,C 180,E1 -26831.81,E2 -26831.81} C_VEL
LIN {X 0,Y 117.515,Z 367.661,A -85,B 0,C 180,E1 -26837.393,E2 -26837.393} C_VEL
LIN {X 0,Y 112.104,Z 370.105,A -85,B 0,C 180,E1 -26842.089,E2 -26842.089} C_VEL
LIN {X 0,Y 107.449,Z 371.635,A -85,B 0,C 180,E1 -26847.242,E2 -26847.242} C_VEL
LIN {X 0,Y 104.279,Z 372.196,A -85,B 0,C 180,E1 -26851.784,E2 -26851.784} C_VEL
LIN {X 0,Y 101.888,Z 372.331,A -85,B 0,C 180,E1 -26854.787,E2 -26854.787} C_VEL
LIN {X 0,Y 96.817,Z 371.952,A -85,B 0,C 180,E1 -26859.703,E2 -26859.703} C_VEL
LIN {X 0,Y 93.124,Z 371.119,A -85,B 0,C 180,E1 -26863.936,E2 -26863.936} C_VEL
LIN {X 0,Y 91.426,Z 370.112,A -85,B 0,C 180,E1 -26867.416,E2 -26867.416} C_VEL
LIN {X 0,Y 91.187,Z 369.664,A -85,B 0,C 180,E1 -26868.624,E2 -26868.624} C_VEL
LIN {X 0,Y 91.081,Z 365.938,A -85,B 0,C 180,E1 -26877.313,E2 -26877.313} C_VEL
LIN {X 0,Y 92.545,Z 360.578,A -85,B 0,C 180,E1 -26885.667,E2 -26885.667} C_VEL
LIN {X 0,Y 94.875,Z 354.338,A -85,B 0,C 180,E1 -26892.769,E2 -26892.769} C_VEL
LIN {X 0,Y 97.739,Z 347.683,A -85,B 0,C 180,E1 -26898.525,E2 -26898.525} C_VEL
LIN {X 0,Y 101.482,Z 339.316,A -85,B 0,C 180,E1 -26904.041,E2 -26904.041} C_VEL
LIN {X 0,Y 105.441,Z 330.295,A -85,B 0,C 180,E1 -26908.566,E2 -26908.566} C_VEL
LIN {X 0,Y 108.834,Z 321.931,A -85,B 0,C 180,E1 -26911.854,E2 -26911.854} C_VEL
LIN {X 0,Y 108.988,Z 317.708,A -85,B 0,C 180,E1 -26913.701,E2 -26913.701} C_VEL
LIN {X 0,Y 108.552,Z 311.264,A -85,B 0,C 180,E1 -26916.499,E2 -26916.499} C_VEL
LIN {X 0,Y 107.558,Z 305.562,A -85,B 0,C 180,E1 -26919.015,E2 -26919.015} C_VEL
LIN {X 0,Y 103.534,Z 295.139,A -85,B 0,C 180,E1 -26924.162,E2 -26924.162} C_VEL
LIN {X 0,Y 100.379,Z 288.916,A -85,B 0,C 180,E1 -26927.551,E2 -26927.551} C_VEL
LIN {X 0,Y 96.083,Z 281.179,A -85,B 0,C 180,E1 -26932.133,E2 -26932.133} C_VEL
LIN {X 0,Y 94.143,Z 278.398,A -85,B 0,C 180,E1 -26934.062,E2 -26934.062} C_VEL
LIN {X 0,Y 93.737,Z 276.813,A -85,B 0,C 180,E1 -26934.86,E2 -26934.86} C_VEL
LIN {X 0,Y 93.59,Z 276.832,A -85,B 0,C 180,E1 -26941.717,E2 -26941.717} C_VEL
LIN {X 0,Y 93.561,Z 276.833,A -85,B 0,C 180,E1 -26946.942,E2 -26946.942} C_VEL
LIN {X 0,Y 93.63,Z 276.824,A -85,B 0,C 180,E1 -26952.503,E2 -26952.503} C_VEL
LIN {X 0,Y 93.627,Z 276.823,A -85,B 0,C 180,E1 -26958.652,E2 -26958.652} C_VEL
LIN {X 0,Y 93.613,Z 276.787,A -85,B 0,C 180,E1 -26965.68,E2 -26965.68} C_VEL
LIN {X 0,Y 93.671,Z 276.813,A -85,B 0,C 180,E1 -26974.213,E2 -26974.213} C_VEL
LIN {X 0,Y 93.696,Z 276.781,A -85,B 0,C 180,E1 -26977.98,E2 -26977.98} C_VEL
LIN {X 0,Y 94.028,Z 276.771,A -85,B 0,C 180,E1 -26986.346,E2 -26986.346} C_VEL
LIN {X 0,Y 94.183,Z 276.73,A -85,B 0,C 180,E1 -26991.424,E2 -26991.424} C_VEL
LIN {X 0,Y 94.797,Z 276.675,A -85,B 0,C 180,E1 -27000.007,E2 -27000.007} C_VEL
LIN {X 0,Y 94.18,Z 276.725,A -85,B 0,C 180,E1 -27008.59,E2 -27008.59} C_VEL
LIN {X 0,Y 94.029,Z 276.774,A -85,B 0,C 180,E1 -27013.657,E2 -27013.657} C_VEL
LIN {X 0,Y 93.704,Z 276.809,A -85,B 0,C 180,E1 -27022.032,E2 -27022.032} C_VEL
LIN {X 0,Y 93.678,Z 276.816,A -85,B 0,C 180,E1 -27026.674,E2 -27026.674} C_VEL
LIN {X 0,Y 94.599,Z 279.517,A -85,B 0,C 180,E1 -27027.824,E2 -27027.824} C_VEL
LIN {X 0,Y 96.87,Z 282.189,A -85,B 0,C 180,E1 -27029.777,E2 -27029.777} C_VEL
LIN {X 0,Y 99.099,Z 287.136,A -85,B 0,C 180,E1 -27032.146,E2 -27032.146} C_VEL
LIN {X 0,Y 102.023,Z 293.943,A -85,B 0,C 180,E1 -27035.241,E2 -27035.241} C_VEL
LIN {X 0,Y 105.231,Z 304.115,A -85,B 0,C 180,E1 -27039.388,E2 -27039.388} C_VEL
LIN {X 0,Y 106.122,Z 307.878,A -85,B 0,C 180,E1 -27040.88,E2 -27040.88} C_VEL
LIN {X 0,Y 106.071,Z 315.057,A -85,B 0,C 180,E1 -27043.206,E2 -27043.206} C_VEL
LIN {X 0,Y 105.373,Z 326.091,A -85,B 0,C 180,E1 -27047.202,E2 -27047.202} C_VEL
LIN {X 0,Y 104.018,Z 337.152,A -85,B 0,C 180,E1 -27051.932,E2 -27051.932} C_VEL
LIN {X 0,Y 102.848,Z 343.574,A -85,B 0,C 180,E1 -27055.095,E2 -27055.095} C_VEL
LIN {X 0,Y 98.825,Z 352.603,A -85,B 0,C 180,E1 -27060.14,E2 -27060.14} C_VEL
LIN {X 0,Y 95.5,Z 360.644,A -85,B 0,C 180,E1 -27066.12,E2 -27066.12} C_VEL
LIN {X 0,Y 93.085,Z 367.073,A -85,B 0,C 180,E1 -27072.418,E2 -27072.418} C_VEL
LIN {X 0,Y 91.786,Z 372.159,A -85,B 0,C 180,E1 -27078.96,E2 -27078.96} C_VEL
LIN {X 0,Y 91.597,Z 376.266,A -85,B 0,C 180,E1 -27085.998,E2 -27085.998} C_VEL
LIN {X 0,Y 91.719,Z 378.03,A -85,B 0,C 180,E1 -27089.996,E2 -27089.996} C_VEL
LIN {X 0,Y 91.412,Z 379.475,A -85,B 0,C 180,E1 -27094.405,E2 -27094.405} C_VEL
LIN {X 0,Y 91.904,Z 381.197,A -85,B 0,C 180,E1 -27103.258,E2 -27103.258} C_VEL
LIN {X 0,Y 94.421,Z 381.416,A -85,B 0,C 180,E1 -27111.844,E2 -27111.844} C_VEL
LIN {X 0,Y 99.162,Z 380.218,A -85,B 0,C 180,E1 -27119.739,E2 -27119.739} C_VEL
LIN {X 0,Y 105.667,Z 377.588,A -85,B 0,C 180,E1 -27126.765,E2 -27126.765} C_VEL
LIN {X 0,Y 113.58,Z 373.384,A -85,B 0,C 180,E1 -27132.889,E2 -27132.889} C_VEL
LIN {X 0,Y 120.411,Z 369.148,A -85,B 0,C 180,E1 -27136.847,E2 -27136.847} C_VEL
LIN {X 0,Y 125.327,Z 365.74,A -85,B 0,C 180,E1 -27139.199,E2 -27139.199} C_VEL
LIN {X 0,Y 127.664,Z 363.872,A -85,B 0,C 180,E1 -27140.412,E2 -27140.412} C_VEL
LIN {X 0,Y 132.701,Z 358.814,A -85,B 0,C 180,E1 -27143.978,E2 -27143.978} C_VEL
LIN {X 0,Y 134.073,Z 357.235,A -85,B 0,C 180,E1 -27145.041,E2 -27145.041} C_VEL
LIN {X 0,Y 135.147,Z 355.71,A -85,B 0,C 180,E1 -27146.304,E2 -27146.304} C_VEL
LIN {X 0,Y 135.961,Z 353.491,A -85,B 0,C 180,E1 -27148.87,E2 -27148.87} C_VEL
LIN {X 0,Y 136.782,Z 350.934,A -85,B 0,C 180,E1 -27152.451,E2 -27152.451} C_VEL
LIN {X 0,Y 137.35,Z 348.489,A -85,B 0,C 180,E1 -27157.07,E2 -27157.07} C_VEL
LIN {X 0,Y 137.724,Z 347.002,A -85,B 0,C 180,E1 -27162.166,E2 -27162.166} C_VEL
LIN {X 0,Y 138.285,Z 346.547,A -85,B 0,C 180,E1 -27168.266,E2 -27168.266} C_VEL
LIN {X 0,Y 138.391,Z 347.034,A -85,B 0,C 180,E1 -27171.232,E2 -27171.232} C_VEL
LIN {X 0,Y 138.108,Z 348.122,A -85,B 0,C 180,E1 -27174.154,E2 -27174.154} C_VEL
LIN {X 0,Y 137.637,Z 349.575,A -85,B 0,C 180,E1 -27177.069,E2 -27177.069} C_VEL
LIN {X 0,Y 136.212,Z 352.617,A -85,B 0,C 180,E1 -27181.474,E2 -27181.474} C_VEL
LIN {X 0,Y 134.752,Z 354.262,A -85,B 0,C 180,E1 -27182.985,E2 -27182.985} C_VEL
LIN {X 0,Y 125.565,Z 361.023,A -85,B 0,C 180,E1 -27187.106,E2 -27187.106} C_VEL
LIN {X 0,Y 117.526,Z 365.802,A -85,B 0,C 180,E1 -27191.467,E2 -27191.467} C_VEL
LIN {X 0,Y 110.063,Z 369.362,A -85,B 0,C 180,E1 -27196.714,E2 -27196.714} C_VEL
LIN {X 0,Y 105.317,Z 371.136,A -85,B 0,C 180,E1 -27200.905,E2 -27200.905} C_VEL
LIN {X 0,Y 101.171,Z 372.216,A -85,B 0,C 180,E1 -27205.446,E2 -27205.446} C_VEL
LIN {X 0,Y 97.609,Z 372.703,A -85,B 0,C 180,E1 -27210.445,E2 -27210.445} C_VEL
LIN {X 0,Y 94.451,Z 372.472,A -85,B 0,C 180,E1 -27216.523,E2 -27216.523} C_VEL
LIN {X 0,Y 92.183,Z 371.274,A -85,B 0,C 180,E1 -27223.317,E2 -27223.317} C_VEL
LIN {X 0,Y 91.187,Z 369.664,A -85,B 0,C 180,E1 -27228.624,E2 -27228.624} C_VEL
LIN {X 0,Y 90.265,Z 368.338,A -85,B 0,C 180,E1 -27232.209,E2 -27232.209} C_VEL
LIN {X 0,Y 87.614,Z 365.527,A -85,B 0,C 180,E1 -27238.1,E2 -27238.1} C_VEL
LIN {X 0,Y 85.883,Z 362.766,A -85,B 0,C 180,E1 -27242.924,E2 -27242.924} C_VEL
LIN {X 0,Y 85.651,Z 360.345,A -85,B 0,C 180,E1 -27246.558,E2 -27246.558} C_VEL
LIN {X 0,Y 85.884,Z 359.471,A -85,B 0,C 180,E1 -27247.739,E2 -27247.739} C_VEL
LIN {X 0,Y 88.509,Z 353.135,A -85,B 0,C 180,E1 -27254.981,E2 -27254.981} C_VEL
LIN {X 0,Y 92.268,Z 344.983,A -85,B 0,C 180,E1 -27261.919,E2 -27261.919} C_VEL
LIN {X 0,Y 95.89,Z 337.341,A -85,B 0,C 180,E1 -27266.823,E2 -27266.823} C_VEL
LIN {X 0,Y 100.216,Z 327.763,A -85,B 0,C 180,E1 -27271.511,E2 -27271.511} C_VEL
LIN {X 0,Y 102.349,Z 322.819,A -85,B 0,C 180,E1 -27273.449,E2 -27273.449} C_VEL
LIN {X 0,Y 102.547,Z 316.937,A -85,B 0,C 180,E1 -27276.217,E2 -27276.217} C_VEL
LIN {X 0,Y 101.69,Z 309.657,A -85,B 0,C 180,E1 -27279.705,E2 -27279.705} C_VEL
LIN {X 0,Y 98.931,Z 301.232,A -85,B 0,C 180,E1 -27284.22,E2 -27284.22} C_VEL
LIN {X 0,Y 96.066,Z 294.753,A -85,B 0,C 180,E1 -27288.024,E2 -27288.024} C_VEL
LIN {X 0,Y 91.814,Z 286.629,A -85,B 0,C 180,E1 -27293.303,E2 -27293.303} C_VEL
LIN {X 0,Y 90.223,Z 284.305,A -85,B 0,C 180,E1 -27295.13,E2 -27295.13} C_VEL
LIN {X 0,Y 89.479,Z 282.582,A -85,B 0,C 180,E1 -27296.218,E2 -27296.218} C_VEL
LIN {X 0,Y 87.187,Z 280.018,A -85,B 0,C 180,E1 -27298.852,E2 -27298.852} C_VEL
LIN {X 0,Y 86.491,Z 277.717,A -85,B 0,C 180,E1 -27300.189,E2 -27300.189} C_VEL
LIN {X 0,Y 86.534,Z 277.709,A -85,B 0,C 180,E1 -27305.705,E2 -27305.705} C_VEL
LIN {X 0,Y 86.557,Z 277.703,A -85,B 0,C 180,E1 -27313.062,E2 -27313.062} C_VEL
LIN {X 0,Y 86.552,Z 277.703,A -85,B 0,C 180,E1 -27319.499,E2 -27319.499} C_VEL
LIN {X 0,Y 86.561,Z 277.664,A -85,B 0,C 180,E1 -27325.375,E2 -27325.375} C_VEL
LIN {X 0,Y 86.587,Z 277.698,A -85,B 0,C 180,E1 -27333.242,E2 -27333.242} C_VEL
LIN {X 0,Y 86.649,Z 277.653,A -85,B 0,C 180,E1 -27341.077,E2 -27341.077} C_VEL
LIN {X 0,Y 86.935,Z 277.653,A -85,B 0,C 180,E1 -27345.972,E2 -27345.972} C_VEL
LIN {X 0,Y 87.092,Z 277.618,A -85,B 0,C 180,E1 -27350.72,E2 -27350.72} C_VEL
LIN {X 0,Y 87.723,Z 277.555,A -85,B 0,C 180,E1 -27360.007,E2 -27360.007} C_VEL
LIN {X 0,Y 87.09,Z 277.61,A -85,B 0,C 180,E1 -27369.295,E2 -27369.295} C_VEL
LIN {X 0,Y 86.941,Z 277.656,A -85,B 0,C 180,E1 -27374.042,E2 -27374.042} C_VEL
LIN {X 0,Y 86.638,Z 277.695,A -85,B 0,C 180,E1 -27381.417,E2 -27381.417} C_VEL
LIN {X 0,Y 87.673,Z 280.597,A -85,B 0,C 180,E1 -27383.011,E2 -27383.011} C_VEL
LIN {X 0,Y 89.752,Z 283.038,A -85,B 0,C 180,E1 -27385.239,E2 -27385.239} C_VEL
LIN {X 0,Y 91.63,Z 286.301,A -85,B 0,C 180,E1 -27387.407,E2 -27387.407} C_VEL
LIN {X 0,Y 92.589,Z 287.475,A -85,B 0,C 180,E1 -27388.328,E2 -27388.328} C_VEL
LIN {X 0,Y 96.72,Z 297.765,A -85,B 0,C 180,E1 -27393.653,E2 -27393.653} C_VEL
LIN {X 0,Y 99.525,Z 307.716,A -85,B 0,C 180,E1 -27398.169,E2 -27398.169} C_VEL
LIN {X 0,Y 100.146,Z 311.403,A -85,B 0,C 180,E1 -27399.702,E2 -27399.702} C_VEL
LIN {X 0,Y 99.268,Z 323.659,A -85,B 0,C 180,E1 -27404.222,E2 -27404.222} C_VEL
LIN {X 0,Y 98.014,Z 333.394,A -85,B 0,C 180,E1 -27408.446,E2 -27408.446} C_VEL
LIN {X 0,Y 96.537,Z 342.313,A -85,B 0,C 180,E1 -27413.017,E2 -27413.017} C_VEL
LIN {X 0,Y 94.257,Z 347.731,A -85,B 0,C 180,E1 -27415.993,E2 -27415.993} C_VEL
LIN {X 0,Y 90.178,Z 356.628,A -85,B 0,C 180,E1 -27422.116,E2 -27422.116} C_VEL
LIN {X 0,Y 87.085,Z 363.776,A -85,B 0,C 180,E1 -27428.701,E2 -27428.701} C_VEL
LIN {X 0,Y 85.16,Z 369.47,A -85,B 0,C 180,E1 -27435.661,E2 -27435.661} C_VEL
LIN {X 0,Y 84.486,Z 373.929,A -85,B 0,C 180,E1 -27442.827,E2 -27442.827} C_VEL
LIN {X 0,Y 84.658,Z 377.232,A -85,B 0,C 180,E1 -27449.995,E2 -27449.995} C_VEL
LIN {X 0,Y 84.349,Z 378.743,A -85,B 0,C 180,E1 -27454.775,E2 -27454.775} C_VEL
LIN {X 0,Y 85.005,Z 380.605,A -85,B 0,C 180,E1 -27464.356,E2 -27464.356} C_VEL
LIN {X 0,Y 87.84,Z 381.036,A -85,B 0,C 180,E1 -27473.576,E2 -27473.576} C_VEL
LIN {X 0,Y 93.036,Z 380.007,A -85,B 0,C 180,E1 -27481.918,E2 -27481.918} C_VEL
LIN {X 0,Y 100.037,Z 377.559,A -85,B 0,C 180,E1 -27489.214,E2 -27489.214} C_VEL
LIN {X 0,Y 106.243,Z 374.728,A -85,B 0,C 180,E1 -27493.988,E2 -27493.988} C_VEL
LIN {X 0,Y 113.204,Z 370.988,A -85,B 0,C 180,E1 -27498.153,E2 -27498.153} C_VEL
LIN {X 0,Y 120.809,Z 366.277,A -85,B 0,C 180,E1 -27501.748,E2 -27501.748} C_VEL
LIN {X 0,Y 123.167,Z 364.53,A -85,B 0,C 180,E1 -27503.015,E2 -27503.015} C_VEL
LIN {X 0,Y 127.373,Z 360.751,A -85,B 0,C 180,E1 -27505.852,E2 -27505.852} C_VEL
LIN {X 0,Y 128.72,Z 359.369,A -85,B 0,C 180,E1 -27506.902,E2 -27506.902} C_VEL
LIN {X 0,Y 130.127,Z 356.962,A -85,B 0,C 180,E1 -27509.778,E2 -27509.778} C_VEL
LIN {X 0,Y 130.987,Z 354.959,A -85,B 0,C 180,E1 -27512.862,E2 -27512.862} C_VEL
LIN {X 0,Y 131.805,Z 352.544,A -85,B 0,C 180,E1 -27518.079,E2 -27518.079} C_VEL
LIN {X 0,Y 132.195,Z 351.326,A -85,B 0,C 180,E1 -27523.115,E2 -27523.115} C_VEL
LIN {X 0,Y 132.642,Z 350.99,A -85,B 0,C 180,E1 -27527.759,E2 -27527.759} C_VEL
LIN {X 0,Y 132.747,Z 351.324,A -85,B 0,C 180,E1 -27530.856,E2 -27530.856} C_VEL
LIN {X 0,Y 132.355,Z 352.275,A -85,B 0,C 180,E1 -27533.899,E2 -27533.899} C_VEL
LIN {X 0,Y 131.643,Z 353.679,A -85,B 0,C 180,E1 -27536.935,E2 -27536.935} C_VEL
LIN {X 0,Y 130.521,Z 355.501,A -85,B 0,C 180,E1 -27539.995,E2 -27539.995} C_VEL
LIN {X 0,Y 129.361,Z 356.623,A -85,B 0,C 180,E1 -27541.057,E2 -27541.057} C_VEL
LIN {X 0,Y 119.948,Z 362.778,A -85,B 0,C 180,E1 -27545.123,E2 -27545.123} C_VEL
LIN {X 0,Y 111.137,Z 367.433,A -85,B 0,C 180,E1 -27549.85,E2 -27549.85} C_VEL
LIN {X 0,Y 102.391,Z 370.926,A -85,B 0,C 180,E1 -27556.082,E2 -27556.082} C_VEL
LIN {X 0,Y 96.958,Z 372.435,A -85,B 0,C 180,E1 -27561.242,E2 -27561.242} C_VEL
LIN {X 0,Y 92.099,Z 373.141,A -85,B 0,C 180,E1 -27567.241,E2 -27567.241} C_VEL
LIN {X 0,Y 88.273,Z 372.932,A -85,B 0,C 180,E1 -27573.861,E2 -27573.861} C_VEL
LIN {X 0,Y 85.304,Z 371.518,A -85,B 0,C 180,E1 -27582.149,E2 -27582.149} C_VEL
LIN {X 0,Y 83.888,Z 368.572,A -85,B 0,C 180,E1 -27591.451,E2 -27591.451} C_VEL
LIN {X 0,Y 84.241,Z 364.557,A -85,B 0,C 180,E1 -27599.968,E2 -27599.968} C_VEL
LIN {X 0,Y 85.884,Z 359.471,A -85,B 0,C 180,E1 -27607.739,E2 -27607.739} C_VEL
LIN {X 0,Y 86.302,Z 356.754,A -85,B 0,C 180,E1 -27611.204,E2 -27611.204} C_VEL
LIN {X 0,Y 85.73,Z 351.773,A -85,B 0,C 180,E1 -27616.912,E2 -27616.912} C_VEL
LIN {X 0,Y 85.71,Z 346.167,A -85,B 0,C 180,E1 -27622.426,E2 -27622.426} C_VEL
LIN {X 0,Y 86.936,Z 342.415,A -85,B 0,C 180,E1 -27625.383,E2 -27625.383} C_VEL
LIN {X 0,Y 91.361,Z 333.46,A -85,B 0,C 180,E1 -27630.822,E2 -27630.822} C_VEL
LIN {X 0,Y 95.945,Z 323.588,A -85,B 0,C 180,E1 -27635.258,E2 -27635.258} C_VEL
LIN {X 0,Y 96.151,Z 317.403,A -85,B 0,C 180,E1 -27638.41,E2 -27638.41} C_VEL
LIN {X 0,Y 95.297,Z 311.154,A -85,B 0,C 180,E1 -27641.799,E2 -27641.799} C_VEL
LIN {X 0,Y 92.407,Z 302.49,A -85,B 0,C 180,E1 -27647.096,E2 -27647.096} C_VEL
LIN {X 0,Y 89.047,Z 295.23,A -85,B 0,C 180,E1 -27652.076,E2 -27652.076} C_VEL
LIN {X 0,Y 87.141,Z 291.35,A -85,B 0,C 180,E1 -27654.962,E2 -27654.962} C_VEL
LIN {X 0,Y 85.098,Z 287.784,A -85,B 0,C 180,E1 -27657.955,E2 -27657.955} C_VEL
LIN {X 0,Y 83.285,Z 285.473,A -85,B 0,C 180,E1 -27660.424,E2 -27660.424} C_VEL
LIN {X 0,Y 82.597,Z 283.746,A -85,B 0,C 180,E1 -27661.708,E2 -27661.708} C_VEL
LIN {X 0,Y 80.227,Z 280.905,A -85,B 0,C 180,E1 -27665.267,E2 -27665.267} C_VEL
LIN {X 0,Y 79.444,Z 278.591,A -85,B 0,C 180,E1 -27667.247,E2 -27667.247} C_VEL
LIN {X 0,Y 79.465,Z 278.579,A -85,B 0,C 180,E1 -27675.042,E2 -27675.042} C_VEL
LIN {X 0,Y 79.452,Z 278.56,A -85,B 0,C 180,E1 -27682.768,E2 -27682.768} C_VEL
LIN {X 0,Y 79.486,Z 278.583,A -85,B 0,C 180,E1 -27692.162,E2 -27692.162} C_VEL
LIN {X 0,Y 79.516,Z 278.539,A -85,B 0,C 180,E1 -27699.305,E2 -27699.305} C_VEL
LIN {X 0,Y 79.829,Z 278.537,A -85,B 0,C 180,E1 -27705.582,E2 -27705.582} C_VEL
LIN {X 0,Y 79.974,Z 278.51,A -85,B 0,C 180,E1 -27709.885,E2 -27709.885} C_VEL
LIN {X 0,Y 80.65,Z 278.436,A -85,B 0,C 180,E1 -27720.008,E2 -27720.008} C_VEL
LIN {X 0,Y 79.974,Z 278.501,A -85,B 0,C 180,E1 -27730.131,E2 -27730.131} C_VEL
LIN {X 0,Y 79.821,Z 278.68,A -85,B 0,C 180,E1 -27734.805,E2 -27734.805} C_VEL
LIN {X 0,Y 80.673,Z 281.349,A -85,B 0,C 180,E1 -27736.59,E2 -27736.59} C_VEL
LIN {X 0,Y 82.716,Z 283.587,A -85,B 0,C 180,E1 -27739.408,E2 -27739.408} C_VEL
LIN {X 0,Y 84.423,Z 286.838,A -85,B 0,C 180,E1 -27742.008,E2 -27742.008} C_VEL
LIN {X 0,Y 86.013,Z 289.181,A -85,B 0,C 180,E1 -27744.121,E2 -27744.121} C_VEL
LIN {X 0,Y 88.598,Z 293.555,A -85,B 0,C 180,E1 -27747.443,E2 -27747.443} C_VEL
LIN {X 0,Y 91.698,Z 302.711,A -85,B 0,C 180,E1 -27752.526,E2 -27752.526} C_VEL
LIN {X 0,Y 93.775,Z 311.222,A -85,B 0,C 180,E1 -27756.846,E2 -27756.846} C_VEL
LIN {X 0,Y 94.042,Z 314.294,A -85,B 0,C 180,E1 -27758.2,E2 -27758.2} C_VEL
LIN {X 0,Y 92.774,Z 325.992,A -85,B 0,C 180,E1 -27762.992,E2 -27762.992} C_VEL
LIN {X 0,Y 91.195,Z 335.566,A -85,B 0,C 180,E1 -27767.592,E2 -27767.592} C_VEL
LIN {X 0,Y 89.877,Z 342.459,A -85,B 0,C 180,E1 -27771.451,E2 -27771.451} C_VEL
LIN {X 0,Y 87.606,Z 347.503,A -85,B 0,C 180,E1 -27774.43,E2 -27774.43} C_VEL
LIN {X 0,Y 83.284,Z 356.351,A -85,B 0,C 180,E1 -27780.968,E2 -27780.968} C_VEL
LIN {X 0,Y 80.044,Z 363.462,A -85,B 0,C 180,E1 -27788.084,E2 -27788.084} C_VEL
LIN {X 0,Y 78.294,Z 368.247,A -85,B 0,C 180,E1 -27794.373,E2 -27794.373} C_VEL
LIN {X 0,Y 77.442,Z 372.88,A -85,B 0,C 180,E1 -27802.171,E2 -27802.171} C_VEL
LIN {X 0,Y 77.603,Z 376.345,A -85,B 0,C 180,E1 -27809.995,E2 -27809.995} C_VEL
LIN {X 0,Y 77.28,Z 377.983,A -85,B 0,C 180,E1 -27815.213,E2 -27815.213} C_VEL
LIN {X 0,Y 78.115,Z 380.011,A -85,B 0,C 180,E1 -27825.654,E2 -27825.654} C_VEL
LIN {X 0,Y 81.356,Z 380.594,A -85,B 0,C 180,E1 -27835.584,E2 -27835.584} C_VEL
LIN {X 0,Y 87.066,Z 379.798,A -85,B 0,C 180,E1 -27844.399,E2 -27844.399} C_VEL
LIN {X 0,Y 94.62,Z 377.521,A -85,B 0,C 180,E1 -27851.944,E2 -27851.944} C_VEL
LIN {X 0,Y 103.63,Z 373.794,A -85,B 0,C 180,E1 -27858.239,E2 -27858.239} C_VEL
LIN {X 0,Y 111.204,Z 369.93,A -85,B 0,C 180,E1 -27862.179,E2 -27862.179} C_VEL
LIN {X 0,Y 116.523,Z 366.832,A -85,B 0,C 180,E1 -27864.506,E2 -27864.506} C_VEL
LIN {X 0,Y 121.167,Z 363.373,A -85,B 0,C 180,E1 -27867.244,E2 -27867.244} C_VEL
LIN {X 0,Y 123.353,Z 361.339,A -85,B 0,C 180,E1 -27869.146,E2 -27869.146} C_VEL
LIN {X 0,Y 124.381,Z 359.844,A -85,B 0,C 180,E1 -27871.291,E2 -27871.291} C_VEL
LIN {X 0,Y 125.113,Z 358.364,A -85,B 0,C 180,E1 -27873.989,E2 -27873.989} C_VEL
LIN {X 0,Y 125.65,Z 357.119,A -85,B 0,C 180,E1 -27876.945,E2 -27876.945} C_VEL
LIN {X 0,Y 126.225,Z 355.862,A -85,B 0,C 180,E1 -27881.169,E2 -27881.169} C_VEL
LIN {X 0,Y 126.468,Z 355.394,A -85,B 0,C 180,E1 -27883.863,E2 -27883.863} C_VEL
LIN {X 0,Y 126.768,Z 355.156,A -85,B 0,C 180,E1 -27887.183,E2 -27887.183} C_VEL
LIN {X 0,Y 126.889,Z 355.3,A -85,B 0,C 180,E1 -27890.43,E2 -27890.43} C_VEL
LIN {X 0,Y 126.38,Z 356.154,A -85,B 0,C 180,E1 -27893.609,E2 -27893.609} C_VEL
LIN {X 0,Y 125.425,Z 357.482,A -85,B 0,C 180,E1 -27896.783,E2 -27896.783} C_VEL
LIN {X 0,Y 124.753,Z 358.286,A -85,B 0,C 180,E1 -27898.381,E2 -27898.381} C_VEL
LIN {X 0,Y 123.538,Z 359.206,A -85,B 0,C 180,E1 -27899.18,E2 -27899.18} C_VEL
LIN {X 0,Y 116.046,Z 363.666,A -85,B 0,C 180,E1 -27902.249,E2 -27902.249} C_VEL
LIN {X 0,Y 106.248,Z 368.396,A -85,B 0,C 180,E1 -27907.19,E2 -27907.19} C_VEL
LIN {X 0,Y 98.421,Z 371.237,A -85,B 0,C 180,E1 -27912.363,E2 -27912.363} C_VEL
LIN {X 0,Y 92.151,Z 372.848,A -85,B 0,C 180,E1 -27917.755,E2 -27917.755} C_VEL
LIN {X 0,Y 85.597,Z 373.587,A -85,B 0,C 180,E1 -27925.435,E2 -27925.435} C_VEL
LIN {X 0,Y 82.132,Z 373.354,A -85,B 0,C 180,E1 -27931.173,E2 -27931.173} C_VEL
LIN {X 0,Y 79.143,Z 372.259,A -85,B 0,C 180,E1 -27938.423,E2 -27938.423} C_VEL
LIN {X 0,Y 77.205,Z 370.124,A -85,B 0,C 180,E1 -27946.726,E2 -27946.726} C_VEL
LIN {X 0,Y 76.864,Z 366.258,A -85,B 0,C 180,E1 -27956.735,E2 -27956.735} C_VEL
LIN {X 0,Y 77.882,Z 362.123,A -85,B 0,C 180,E1 -27964.454,E2 -27964.454} C_VEL
LIN {X 0,Y 79.83,Z 357.127,A -85,B 0,C 180,E1 -27971.6,E2 -27971.6} C_VEL
LIN {X 0,Y 83.004,Z 350.268,A -85,B 0,C 180,E1 -27979.023,E2 -27979.023} C_VEL
LIN {X 0,Y 86.936,Z 342.415,A -85,B 0,C 180,E1 -27985.383,E2 -27985.383} C_VEL
LIN {X 0,Y 88.882,Z 337.117,A -85,B 0,C 180,E1 -27989.021,E2 -27989.021} C_VEL
LIN {X 0,Y 89.857,Z 331.543,A -85,B 0,C 180,E1 -27992.647,E2 -27992.647} C_VEL
LIN {X 0,Y 90.13,Z 325.829,A -85,B 0,C 180,E1 -27996.245,E2 -27996.245} C_VEL
LIN {X 0,Y 89.904,Z 319.972,A -85,B 0,C 180,E1 -27999.755,E2 -27999.755} C_VEL
LIN {X 0,Y 89.486,Z 315.214,A -85,B 0,C 180,E1 -28002.577,E2 -28002.577} C_VEL
LIN {X 0,Y 87.335,Z 307.715,A -85,B 0,C 180,E1 -28007.593,E2 -28007.593} C_VEL
LIN {X 0,Y 84.214,Z 300.023,A -85,B 0,C 180,E1 -28013.386,E2 -28013.386} C_VEL
LIN {X 0,Y 81.518,Z 294.397,A -85,B 0,C 180,E1 -28018.238,E2 -28018.238} C_VEL
LIN {X 0,Y 78.404,Z 289.003,A -85,B 0,C 180,E1 -28023.806,E2 -28023.806} C_VEL
LIN {X 0,Y 76.984,Z 287.143,A -85,B 0,C 180,E1 -28026.391,E2 -28026.391} C_VEL
LIN {X 0,Y 75.931,Z 284.787,A -85,B 0,C 180,E1 -28028.901,E2 -28028.901} C_VEL
LIN {X 0,Y 74.62,Z 283.896,A -85,B 0,C 180,E1 -28031.253,E2 -28031.253} C_VEL
LIN {X 0,Y 72.704,Z 280.925,A -85,B 0,C 180,E1 -28036.047,E2 -28036.047} C_VEL
LIN {X 0,Y 72.303,Z 279.478,A -85,B 0,C 180,E1 -28037.961,E2 -28037.961} C_VEL
LIN {X 0,Y 72.338,Z 279.435,A -85,B 0,C 180,E1 -28044.354,E2 -28044.354} C_VEL
LIN {X 0,Y 72.393,Z 279.462,A -85,B 0,C 180,E1 -28050.971,E2 -28050.971} C_VEL
LIN {X 0,Y 72.397,Z 279.434,A -85,B 0,C 180,E1 -28057.161,E2 -28057.161} C_VEL
LIN {X 0,Y 72.726,Z 279.417,A -85,B 0,C 180,E1 -28065.119,E2 -28065.119} C_VEL
LIN {X 0,Y 72.864,Z 279.402,A -85,B 0,C 180,E1 -28068.886,E2 -28068.886} C_VEL
LIN {X 0,Y 73.576,Z 279.317,A -85,B 0,C 180,E1 -28080.008,E2 -28080.008} C_VEL
LIN {X 0,Y 73.076,Z 279.358,A -85,B 0,C 180,E1 -28085.009,E2 -28085.009} C_VEL
LIN {X 0,Y 73.659,Z 281.661,A -85,B 0,C 180,E1 -28087.202,E2 -28087.202} C_VEL
LIN {X 0,Y 75.618,Z 284.191,A -85,B 0,C 180,E1 -28091.441,E2 -28091.441} C_VEL
LIN {X 0,Y 76.465,Z 284.94,A -85,B 0,C 180,E1 -28092.921,E2 -28092.921} C_VEL
LIN {X 0,Y 77.738,Z 287.911,A -85,B 0,C 180,E1 -28095.745,E2 -28095.745} C_VEL
LIN {X 0,Y 79.623,Z 290.593,A -85,B 0,C 180,E1 -28098.886,E2 -28098.886} C_VEL
LIN {X 0,Y 83.38,Z 297.258,A -85,B 0,C 180,E1 -28104.934,E2 -28104.934} C_VEL
LIN {X 0,Y 84.585,Z 300.56,A -85,B 0,C 180,E1 -28107.2,E2 -28107.2} C_VEL
LIN {X 0,Y 86.8,Z 308.467,A -85,B 0,C 180,E1 -28111.957,E2 -28111.957} C_VEL
LIN {X 0,Y 87.995,Z 314.654,A -85,B 0,C 180,E1 -28115.391,E2 -28115.391} C_VEL
LIN {X 0,Y 87.69,Z 318.898,A -85,B 0,C 180,E1 -28117.274,E2 -28117.274} C_VEL
LIN {X 0,Y 85.944,Z 330.22,A -85,B 0,C 180,E1 -28122.604,E2 -28122.604} C_VEL
LIN {X 0,Y 83.604,Z 341.272,A -85,B 0,C 180,E1 -28128.88,E2 -28128.88} C_VEL
LIN {X 0,Y 82.608,Z 344.218,A -85,B 0,C 180,E1 -28130.739,E2 -28130.739} C_VEL
LIN {X 0,Y 77.798,Z 353.3,A -85,B 0,C 180,E1 -28137.173,E2 -28137.173} C_VEL
LIN {X 0,Y 74.01,Z 360.914,A -85,B 0,C 180,E1 -28144.696,E2 -28144.696} C_VEL
LIN {X 0,Y 71.483,Z 366.999,A -85,B 0,C 180,E1 -28152.84,E2 -28152.84} C_VEL
LIN {X 0,Y 70.4,Z 371.808,A -85,B 0,C 180,E1 -28161.382,E2 -28161.382} C_VEL
LIN {X 0,Y 70.439,Z 374.018,A -85,B 0,C 180,E1 -28166.269,E2 -28166.269} C_VEL
LIN {X 0,Y 70.547,Z 375.449,A -85,B 0,C 180,E1 -28169.994,E2 -28169.994} C_VEL
LIN {X 0,Y 70.238,Z 377.162,A -85,B 0,C 180,E1 -28175.737,E2 -28175.737} C_VEL
LIN {X 0,Y 71.285,Z 379.399,A -85,B 0,C 180,E1 -28187.198,E2 -28187.198} C_VEL
LIN {X 0,Y 74.991,Z 380.149,A -85,B 0,C 180,E1 -28197.937,E2 -28197.937} C_VEL
LIN {X 0,Y 81.287,Z 379.521,A -85,B 0,C 180,E1 -28207.238,E2 -28207.238} C_VEL
LIN {X 0,Y 89.454,Z 377.503,A -85,B 0,C 180,E1 -28214.992,E2 -28214.992} C_VEL
LIN {X 0,Y 99.037,Z 373.97,A -85,B 0,C 180,E1 -28221.309,E2 -28221.309} C_VEL
LIN {X 0,Y 107.014,Z 370.297,A -85,B 0,C 180,E1 -28225.17,E2 -28225.17} C_VEL
LIN {X 0,Y 112.5,Z 367.318,A -85,B 0,C 180,E1 -28227.49,E2 -28227.49} C_VEL
LIN {X 0,Y 114.974,Z 365.744,A -85,B 0,C 180,E1 -28228.839,E2 -28228.839} C_VEL
LIN {X 0,Y 116.673,Z 364.503,A -85,B 0,C 180,E1 -28229.973,E2 -28229.973} C_VEL
LIN {X 0,Y 117.916,Z 363.353,A -85,B 0,C 180,E1 -28231.517,E2 -28231.517} C_VEL
LIN {X 0,Y 118.489,Z 362.597,A -85,B 0,C 180,E1 -28232.828,E2 -28232.828} C_VEL
LIN {X 0,Y 119.187,Z 361.346,A -85,B 0,C 180,E1 -28235.616,E2 -28235.616} C_VEL
LIN {X 0,Y 119.902,Z 360.059,A -85,B 0,C 180,E1 -28239.68,E2 -28239.68} C_VEL
LIN {X 0,Y 120.349,Z 359.332,A -85,B 0,C 180,E1 -28243.018,E2 -28243.018} C_VEL
LIN {X 0,Y 120.672,Z 358.985,A -85,B 0,C 180,E1 -28246.523,E2 -28246.523} C_VEL
LIN {X 0,Y 120.813,Z 359,A -85,B 0,C 180,E1 -28249.944,E2 -28249.944} C_VEL
LIN {X 0,Y 120.214,Z 359.738,A -85,B 0,C 180,E1 -28253.28,E2 -28253.28} C_VEL
LIN {X 0,Y 119.034,Z 360.946,A -85,B 0,C 180,E1 -28256.61,E2 -28256.61} C_VEL
LIN {X 0,Y 110.52,Z 365.499,A -85,B 0,C 180,E1 -28259.994,E2 -28259.994} C_VEL
LIN {X 0,Y 102.22,Z 369.095,A -85,B 0,C 180,E1 -28263.936,E2 -28263.936} C_VEL
LIN {X 0,Y 92.727,Z 372.157,A -85,B 0,C 180,E1 -28269.864,E2 -28269.864} C_VEL
LIN {X 0,Y 87.099,Z 373.37,A -85,B 0,C 180,E1 -28274.49,E2 -28274.49} C_VEL
LIN {X 0,Y 81.706,Z 374.002,A -85,B 0,C 180,E1 -28280.116,E2 -28280.116} C_VEL
LIN {X 0,Y 76.678,Z 373.83,A -85,B 0,C 180,E1 -28287.267,E2 -28287.267} C_VEL
LIN {X 0,Y 72.861,Z 372.734,A -85,B 0,C 180,E1 -28295.351,E2 -28295.351} C_VEL
LIN {X 0,Y 70.256,Z 370.291,A -85,B 0,C 180,E1 -28305.562,E2 -28305.562} C_VEL
LIN {X 0,Y 69.789,Z 366.144,A -85,B 0,C 180,E1 -28316.88,E2 -28316.88} C_VEL
LIN {X 0,Y 71.205,Z 361.066,A -85,B 0,C 180,E1 -28326.753,E2 -28326.753} C_VEL
LIN {X 0,Y 73.771,Z 355.256,A -85,B 0,C 180,E1 -28335.092,E2 -28335.092} C_VEL
LIN {X 0,Y 76.775,Z 349.316,A -85,B 0,C 180,E1 -28341.551,E2 -28341.551} C_VEL
LIN {X 0,Y 81.504,Z 340.423,A -85,B 0,C 180,E1 -28348.77,E2 -28348.77} C_VEL
LIN {X 0,Y 86.751,Z 330.282,A -85,B 0,C 180,E1 -28354.652,E2 -28354.652} C_VEL
LIN {X 0,Y 89.614,Z 324.33,A -85,B 0,C 180,E1 -28357.326,E2 -28357.326} C_VEL
LIN {X 0,Y 89.904,Z 319.972,A -85,B 0,C 180,E1 -28359.755,E2 -28359.755} C_VEL
LIN {X 0,Y 89.357,Z 317.251,A -85,B 0,C 180,E1 -28361.526,E2 -28361.526} C_VEL
LIN {X 0,Y 88.219,Z 314.873,A -85,B 0,C 180,E1 -28363.41,E2 -28363.41} C_VEL
LIN {X 0,Y 84.902,Z 310.887,A -85,B 0,C 180,E1 -28367.416,E2 -28367.416} C_VEL
LIN {X 0,Y 79.742,Z 305.207,A -85,B 0,C 180,E1 -28374.152,E2 -28374.152} C_VEL
LIN {X 0,Y 78.535,Z 302.937,A -85,B 0,C 180,E1 -28376.464,E2 -28376.464} C_VEL
LIN {X 0,Y 76.468,Z 298.458,A -85,B 0,C 180,E1 -28380.929,E2 -28380.929} C_VEL
LIN {X 0,Y 74.591,Z 294.83,A -85,B 0,C 180,E1 -28385.127,E2 -28385.127} C_VEL
LIN {X 0,Y 72.832,Z 291.611,A -85,B 0,C 180,E1 -28389.483,E2 -28389.483} C_VEL
LIN {X 0,Y 69.925,Z 287.331,A -85,B 0,C 180,E1 -28397.366,E2 -28397.366} C_VEL
LIN {X 0,Y 69.546,Z 286.147,A -85,B 0,C 180,E1 -28399.095,E2 -28399.095} C_VEL
LIN {X 0,Y 66.262,Z 283.145,A -85,B 0,C 180,E1 -28415.743,E2 -28415.743} C_VEL
LIN {X 0,Y 66.219,Z 282.665,A -85,B 0,C 180,E1 -28422.803,E2 -28422.803} C_VEL
LIN {X 0,Y 66.882,Z 283.21,A -85,B 0,C 180,E1 -28430.178,E2 -28430.178} C_VEL
LIN {X 0,Y 69.558,Z 285.299,A -85,B 0,C 180,E1 -28441.203,E2 -28441.203} C_VEL
LIN {X 0,Y 73.063,Z 290.923,A -85,B 0,C 180,E1 -28451.1,E2 -28451.1} C_VEL
LIN {X 0,Y 74.068,Z 293.461,A -85,B 0,C 180,E1 -28453.903,E2 -28453.903} C_VEL
LIN {X 0,Y 76.034,Z 296.795,A -85,B 0,C 180,E1 -28457.951,E2 -28457.951} C_VEL
LIN {X 0,Y 78.969,Z 302.553,A -85,B 0,C 180,E1 -28463.617,E2 -28463.617} C_VEL
LIN {X 0,Y 80.854,Z 310.006,A -85,B 0,C 180,E1 -28468.852,E2 -28468.852} C_VEL
LIN {X 0,Y 81.987,Z 316.794,A -85,B 0,C 180,E1 -28473.134,E2 -28473.134} C_VEL
LIN {X 0,Y 81.885,Z 319.158,A -85,B 0,C 180,E1 -28474.331,E2 -28474.331} C_VEL
LIN {X 0,Y 79.949,Z 329.846,A -85,B 0,C 180,E1 -28479.712,E2 -28479.712} C_VEL
LIN {X 0,Y 77.464,Z 340.071,A -85,B 0,C 180,E1 -28485.866,E2 -28485.866} C_VEL
LIN {X 0,Y 76.126,Z 344.099,A -85,B 0,C 180,E1 -28488.607,E2 -28488.607} C_VEL
LIN {X 0,Y 71.114,Z 352.982,A -85,B 0,C 180,E1 -28495.365,E2 -28495.365} C_VEL
LIN {X 0,Y 67.049,Z 360.564,A -85,B 0,C 180,E1 -28503.539,E2 -28503.539} C_VEL
LIN {X 0,Y 64.104,Z 367.514,A -85,B 0,C 180,E1 -28514.086,E2 -28514.086} C_VEL
LIN {X 0,Y 63.3,Z 372.105,A -85,B 0,C 180,E1 -28523.619,E2 -28523.619} C_VEL
LIN {X 0,Y 63.478,Z 374.523,A -85,B 0,C 180,E1 -28529.994,E2 -28529.994} C_VEL
LIN {X 0,Y 63.2,Z 376.31,A -85,B 0,C 180,E1 -28536.378,E2 -28536.378} C_VEL
LIN {X 0,Y 64.528,Z 378.717,A -85,B 0,C 180,E1 -28549.064,E2 -28549.064} C_VEL
LIN {X 0,Y 68.78,Z 379.698,A -85,B 0,C 180,E1 -28560.717,E2 -28560.717} C_VEL
LIN {X 0,Y 75.741,Z 379.249,A -85,B 0,C 180,E1 -28570.499,E2 -28570.499} C_VEL
LIN {X 0,Y 84.574,Z 377.416,A -85,B 0,C 180,E1 -28578.4,E2 -28578.4} C_VEL
LIN {X 0,Y 94.764,Z 374.152,A -85,B 0,C 180,E1 -28584.658,E2 -28584.658} C_VEL
LIN {X 0,Y 103.141,Z 370.677,A -85,B 0,C 180,E1 -28588.394,E2 -28588.394} C_VEL
LIN {X 0,Y 108.787,Z 367.861,A -85,B 0,C 180,E1 -28590.701,E2 -28590.701} C_VEL
LIN {X 0,Y 111.247,Z 366.351,A -85,B 0,C 180,E1 -28592.175,E2 -28592.175} C_VEL
LIN {X 0,Y 112.317,Z 365.36,A -85,B 0,C 180,E1 -28594.017,E2 -28594.017} C_VEL
LIN {X 0,Y 113.335,Z 363.848,A -85,B 0,C 180,E1 -28598.45,E2 -28598.45} C_VEL
LIN {X 0,Y 113.939,Z 362.995,A -85,B 0,C 180,E1 -28602.031,E2 -28602.031} C_VEL
LIN {X 0,Y 114.352,Z 362.51,A -85,B 0,C 180,E1 -28605.763,E2 -28605.763} C_VEL
LIN {X 0,Y 114.541,Z 362.413,A -85,B 0,C 180,E1 -28609.387,E2 -28609.387} C_VEL
LIN {X 0,Y 113.877,Z 363.015,A -85,B 0,C 180,E1 -28612.904,E2 -28612.904} C_VEL
LIN {X 0,Y 112.944,Z 363.637,A -85,B 0,C 180,E1 -28614.587,E2 -28614.587} C_VEL
LIN {X 0,Y 102.217,Z 368.467,A -85,B 0,C 180,E1 -28618.741,E2 -28618.741} C_VEL
LIN {X 0,Y 91.325,Z 372.048,A -85,B 0,C 180,E1 -28624.407,E2 -28624.407} C_VEL
LIN {X 0,Y 83.746,Z 373.702,A -85,B 0,C 180,E1 -28629.655,E2 -28629.655} C_VEL
LIN {X 0,Y 77.063,Z 374.437,A -85,B 0,C 180,E1 -28635.87,E2 -28635.87} C_VEL
LIN {X 0,Y 69.994,Z 374.077,A -85,B 0,C 180,E1 -28645.367,E2 -28645.367} C_VEL
LIN {X 0,Y 66.56,Z 373.101,A -85,B 0,C 180,E1 -28652.371,E2 -28652.371} C_VEL
LIN {X 0,Y 63.846,Z 371.162,A -85,B 0,C 180,E1 -28661.321,E2 -28661.321} C_VEL
LIN {X 0,Y 62.599,Z 368.008,A -85,B 0,C 180,E1 -28671.786,E2 -28671.786} C_VEL
LIN {X 0,Y 63.389,Z 363.049,A -85,B 0,C 180,E1 -28683.681,E2 -28683.681} C_VEL
LIN {X 0,Y 65.883,Z 357.202,A -85,B 0,C 180,E1 -28693.717,E2 -28693.717} C_VEL
LIN {X 0,Y 69.744,Z 349.948,A -85,B 0,C 180,E1 -28702.77,E2 -28702.77} C_VEL
LIN {X 0,Y 74.326,Z 341.917,A -85,B 0,C 180,E1 -28710.005,E2 -28710.005} C_VEL
LIN {X 0,Y 79.799,Z 332.029,A -85,B 0,C 180,E1 -28716.326,E2 -28716.326} C_VEL
LIN {X 0,Y 83.41,Z 325.042,A -85,B 0,C 180,E1 -28719.707,E2 -28719.707} C_VEL
LIN {X 0,Y 83.61,Z 320.568,A -85,B 0,C 180,E1 -28722.498,E2 -28722.498} C_VEL
LIN {X 0,Y 83.254,Z 317.33,A -85,B 0,C 180,E1 -28724.675,E2 -28724.675} C_VEL
LIN {X 0,Y 81.302,Z 309.99,A -85,B 0,C 180,E1 -28730.234,E2 -28730.234} C_VEL
LIN {X 0,Y 78.535,Z 302.937,A -85,B 0,C 180,E1 -28736.464,E2 -28736.464} C_VEL
LIN {X 0,Y 77.328,Z 300.915,A -85,B 0,C 180,E1 -28738.77,E2 -28738.77} C_VEL
LIN {X 0,Y 74.884,Z 298.874,A -85,B 0,C 180,E1 -28742.534,E2 -28742.534} C_VEL
LIN {X 0,Y 68.897,Z 296.074,A -85,B 0,C 180,E1 -28752.55,E2 -28752.55} C_VEL
LIN {X 0,Y 67.219,Z 294.341,A -85,B 0,C 180,E1 -28757.259,E2 -28757.259} C_VEL
LIN {X 0,Y 66.889,Z 293.534,A -85,B 0,C 180,E1 -28758.825,E2 -28758.825} C_VEL
LIN {X 0,Y 66.562,Z 292.475,A -85,B 0,C 180,E1 -28760.703,E2 -28760.703} C_VEL
LIN {X 0,Y 64.175,Z 290.172,A -85,B 0,C 180,E1 -28774.032,E2 -28774.032} C_VEL
LIN {X 0,Y 64.068,Z 289.536,A -85,B 0,C 180,E1 -28780.797,E2 -28780.797} C_VEL
LIN {X 0,Y 64.569,Z 289.709,A -85,B 0,C 180,E1 -28788.44,E2 -28788.44} C_VEL
LIN {X 0,Y 66.894,Z 291.72,A -85,B 0,C 180,E1 -28800.009,E2 -28800.009} C_VEL
LIN {X 0,Y 69.308,Z 296.462,A -85,B 0,C 180,E1 -28808.758,E2 -28808.758} C_VEL
LIN {X 0,Y 72.196,Z 302.745,A -85,B 0,C 180,E1 -28816.989,E2 -28816.989} C_VEL
LIN {X 0,Y 74.304,Z 307.747,A -85,B 0,C 180,E1 -28822.239,E2 -28822.239} C_VEL
LIN {X 0,Y 75.637,Z 314.839,A -85,B 0,C 180,E1 -28827.692,E2 -28827.692} C_VEL
LIN {X 0,Y 76.15,Z 319.986,A -85,B 0,C 180,E1 -28831.281,E2 -28831.281} C_VEL
LIN {X 0,Y 73.78,Z 330.741,A -85,B 0,C 180,E1 -28837.18,E2 -28837.18} C_VEL
LIN {X 0,Y 70.881,Z 341.032,A -85,B 0,C 180,E1 -28843.964,E2 -28843.964} C_VEL
LIN {X 0,Y 70.206,Z 343.057,A -85,B 0,C 180,E1 -28845.506,E2 -28845.506} C_VEL
LIN {X 0,Y 64.509,Z 352.561,A -85,B 0,C 180,E1 -28853.179,E2 -28853.179} C_VEL
LIN {X 0,Y 60.124,Z 360.134,A -85,B 0,C 180,E1 -28862.116,E2 -28862.116} C_VEL
LIN {X 0,Y 57.293,Z 366.195,A -85,B 0,C 180,E1 -28872.134,E2 -28872.134} C_VEL
LIN {X 0,Y 56.255,Z 370.984,A -85,B 0,C 180,E1 -28882.816,E2 -28882.816} C_VEL
LIN {X 0,Y 56.416,Z 373.521,A -85,B 0,C 180,E1 -28889.993,E2 -28889.993} C_VEL
LIN {X 0,Y 56.168,Z 375.448,A -85,B 0,C 180,E1 -28897.181,E2 -28897.181} C_VEL
LIN {X 0,Y 57.862,Z 378.021,A -85,B 0,C 180,E1 -28911.362,E2 -28911.362} C_VEL
LIN {X 0,Y 62.769,Z 379.171,A -85,B 0,C 180,E1 -28924.036,E2 -28924.036} C_VEL
LIN {X 0,Y 70.479,Z 378.969,A -85,B 0,C 180,E1 -28934.26,E2 -28934.26} C_VEL
LIN {X 0,Y 80.018,Z 377.328,A -85,B 0,C 180,E1 -28942.221,E2 -28942.221} C_VEL
LIN {X 0,Y 90.836,Z 374.287,A -85,B 0,C 180,E1 -28948.32,E2 -28948.32} C_VEL
LIN {X 0,Y 99.612,Z 370.997,A -85,B 0,C 180,E1 -28951.866,E2 -28951.866} C_VEL
LIN {X 0,Y 102.603,Z 369.718,A -85,B 0,C 180,E1 -28952.922,E2 -28952.922} C_VEL
LIN {X 0,Y 105.054,Z 368.497,A -85,B 0,C 180,E1 -28954.053,E2 -28954.053} C_VEL
LIN {X 0,Y 106.529,Z 367.229,A -85,B 0,C 180,E1 -28957.45,E2 -28957.45} C_VEL
LIN {X 0,Y 107.246,Z 366.373,A -85,B 0,C 180,E1 -28960.868,E2 -28960.868} C_VEL
LIN {X 0,Y 107.817,Z 365.734,A -85,B 0,C 180,E1 -28964.88,E2 -28964.88} C_VEL
LIN {X 0,Y 108.085,Z 365.52,A -85,B 0,C 180,E1 -28968.745,E2 -28968.745} C_VEL
LIN {X 0,Y 106.601,Z 366.261,A -85,B 0,C 180,E1 -28972.417,E2 -28972.417} C_VEL
LIN {X 0,Y 97.272,Z 369.901,A -85,B 0,C 180,E1 -28975.85,E2 -28975.85} C_VEL
LIN {X 0,Y 88.497,Z 372.487,A -85,B 0,C 180,E1 -28979.993,E2 -28979.993} C_VEL
LIN {X 0,Y 77.85,Z 374.446,A -85,B 0,C 180,E1 -28986.812,E2 -28986.812} C_VEL
LIN {X 0,Y 71.872,Z 374.901,A -85,B 0,C 180,E1 -28992.108,E2 -28992.108} C_VEL
LIN {X 0,Y 66.428,Z 374.723,A -85,B 0,C 180,E1 -28998.495,E2 -28998.495} C_VEL
LIN {X 0,Y 61.128,Z 373.666,A -85,B 0,C 180,E1 -29007.368,E2 -29007.368} C_VEL
LIN {X 0,Y 57.432,Z 371.65,A -85,B 0,C 180,E1 -29017.71,E2 -29017.71} C_VEL
LIN {X 0,Y 55.551,Z 368.109,A -85,B 0,C 180,E1 -29030.77,E2 -29030.77} C_VEL
LIN {X 0,Y 55.935,Z 364.159,A -85,B 0,C 180,E1 -29041.561,E2 -29041.561} C_VEL
LIN {X 0,Y 57.853,Z 359.422,A -85,B 0,C 180,E1 -29051.372,E2 -29051.372} C_VEL
LIN {X 0,Y 61.555,Z 352.596,A -85,B 0,C 180,E1 -29061.802,E2 -29061.802} C_VEL
LIN {X 0,Y 66.109,Z 345.001,A -85,B 0,C 180,E1 -29070.006,E2 -29070.006} C_VEL
LIN {X 0,Y 71.722,Z 335.666,A -85,B 0,C 180,E1 -29077.106,E2 -29077.106} C_VEL
LIN {X 0,Y 76.759,Z 326.792,A -85,B 0,C 180,E1 -29081.894,E2 -29081.894} C_VEL
LIN {X 0,Y 77.313,Z 325.638,A -85,B 0,C 180,E1 -29082.473,E2 -29082.473} C_VEL
LIN {X 0,Y 77.366,Z 320.996,A -85,B 0,C 180,E1 -29085.82,E2 -29085.82} C_VEL
LIN {X 0,Y 75.762,Z 313.816,A -85,B 0,C 180,E1 -29091.954,E2 -29091.954} C_VEL
LIN {X 0,Y 72.978,Z 305.749,A -85,B 0,C 180,E1 -29099.939,E2 -29099.939} C_VEL
LIN {X 0,Y 70.428,Z 300.131,A -85,B 0,C 180,E1 -29107.045,E2 -29107.045} C_VEL
LIN {X 0,Y 68.8,Z 296.914,A -85,B 0,C 180,E1 -29111.98,E2 -29111.98} C_VEL
LIN {X 0,Y 66.889,Z 293.534,A -85,B 0,C 180,E1 -29118.825,E2 -29118.825} C_VEL
LIN {X 0,Y 66.219,Z 292.312,A -85,B 0,C 180,E1 -29121.947,E2 -29121.947} C_VEL
LIN {X 0,Y 64.908,Z 291.893,A -85,B 0,C 180,E1 -29126.947,E2 -29126.947} C_VEL
LIN {X 0,Y 63.593,Z 292.635,A -85,B 0,C 180,E1 -29132.093,E2 -29132.093} C_VEL
LIN {X 0,Y 61.926,Z 296.267,A -85,B 0,C 180,E1 -29146.989,E2 -29146.989} C_VEL
LIN {X 0,Y 63.366,Z 297.763,A -85,B 0,C 180,E1 -29156.67,E2 -29156.67} C_VEL
LIN {X 0,Y 64.067,Z 298.691,A -85,B 0,C 180,E1 -29160.01,E2 -29160.01} C_VEL
LIN {X 0,Y 65.381,Z 301.821,A -85,B 0,C 180,E1 -29166.18,E2 -29166.18} C_VEL
LIN {X 0,Y 67.798,Z 307.759,A -85,B 0,C 180,E1 -29175.029,E2 -29175.029} C_VEL
LIN {X 0,Y 69.45,Z 312.76,A -85,B 0,C 180,E1 -29180.753,E2 -29180.753} C_VEL
LIN {X 0,Y 70.252,Z 319.92,A -85,B 0,C 180,E1 -29186.761,E2 -29186.761} C_VEL
LIN {X 0,Y 70.344,Z 321.97,A -85,B 0,C 180,E1 -29188.339,E2 -29188.339} C_VEL
LIN {X 0,Y 67.845,Z 331.377,A -85,B 0,C 180,E1 -29194.023,E2 -29194.023} C_VEL
LIN {X 0,Y 64.807,Z 340.599,A -85,B 0,C 180,E1 -29200.604,E2 -29200.604} C_VEL
LIN {X 0,Y 64.109,Z 342.59,A -85,B 0,C 180,E1 -29202.262,E2 -29202.262} C_VEL
LIN {X 0,Y 59.941,Z 349.2,A -85,B 0,C 180,E1 -29207.6,E2 -29207.6} C_VEL
LIN {X 0,Y 54.7,Z 357.355,A -85,B 0,C 180,E1 -29216.895,E2 -29216.895} C_VEL
LIN {X 0,Y 51.465,Z 362.901,A -85,B 0,C 180,E1 -29225.807,E2 -29225.807} C_VEL
LIN {X 0,Y 49.428,Z 368.309,A -85,B 0,C 180,E1 -29237.677,E2 -29237.677} C_VEL
LIN {X 0,Y 49.384,Z 372.492,A -85,B 0,C 180,E1 -29249.992,E2 -29249.992} C_VEL
LIN {X 0,Y 49.17,Z 374.493,A -85,B 0,C 180,E1 -29258.209,E2 -29258.209} C_VEL
LIN {X 0,Y 51.318,Z 377.306,A -85,B 0,C 180,E1 -29274.249,E2 -29274.249} C_VEL
LIN {X 0,Y 57.016,Z 378.637,A -85,B 0,C 180,E1 -29288.039,E2 -29288.039} C_VEL
LIN {X 0,Y 65.571,Z 378.617,A -85,B 0,C 180,E1 -29298.605,E2 -29298.605} C_VEL
LIN {X 0,Y 75.857,Z 377.238,A -85,B 0,C 180,E1 -29306.484,E2 -29306.484} C_VEL
